LIN {X 0,Y 150.683,Z 393.041,A -85,B 0,C 180,E1 7413.083,E2 7413.083} C_VEL
LIN {X 0,Y 146.558,Z 378.59,A -85,B 0,C 180,E1 7406.767,E2 7406.767} C_VEL
LIN {X 0,Y 142.773,Z 366.039,A -85,B 0,C 180,E1 7400.503,E2 7400.503} C_VEL
LIN {X 0,Y 139.358,Z 355.664,A -85,B 0,C 180,E1 7394.549,E2 7394.549} C_VEL
LIN {X 0,Y 136.525,Z 347.614,A -85,B 0,C 180,E1 7389.278,E2 7389.278} C_VEL
LIN {X 0,Y 133.958,Z 340.934,A -85,B 0,C 180,E1 7384.287,E2 7384.287} C_VEL
LIN {X 0,Y 132.496,Z 337.338,A -85,B 0,C 180,E1 7381.303,E2 7381.303} C_VEL
LIN {X 0,Y 131.528,Z 334.4,A -85,B 0,C 180,E1 7378.699,E2 7378.699} C_VEL
LIN {X 0,Y 131.538,Z 334.397,A -85,B 0,C 180,E1 7371.703,E2 7371.703} C_VEL
LIN {X 0,Y 131.537,Z 334.414,A -85,B 0,C 180,E1 7364.864,E2 7364.864} C_VEL
LIN {X 0,Y 131.54,Z 334.399,A -85,B 0,C 180,E1 7358.015,E2 7358.015} C_VEL
LIN {X 0,Y 131.539,Z 334.371,A -85,B 0,C 180,E1 7350.936,E2 7350.936} C_VEL
LIN {X 0,Y 131.536,Z 334.411,A -85,B 0,C 180,E1 7344.184,E2 7344.184} C_VEL
LIN {X 0,Y 131.542,Z 334.371,A -85,B 0,C 180,E1 7337.439,E2 7337.439} C_VEL
LIN {X 0,Y 131.54,Z 334.396,A -85,B 0,C 180,E1 7330.537,E2 7330.537} C_VEL
LIN {X 0,Y 131.548,Z 334.386,A -85,B 0,C 180,E1 7323.696,E2 7323.696} C_VEL
LIN {X 0,Y 131.551,Z 334.382,A -85,B 0,C 180,E1 7317.128,E2 7317.128} C_VEL
LIN {X 0,Y 131.548,Z 334.403,A -85,B 0,C 180,E1 7310.461,E2 7310.461} C_VEL
LIN {X 0,Y 131.548,Z 334.375,A -85,B 0,C 180,E1 7303.625,E2 7303.625} C_VEL
LIN {X 0,Y 131.549,Z 334.398,A -85,B 0,C 180,E1 7296.543,E2 7296.543} C_VEL
LIN {X 0,Y 131.56,Z 334.411,A -85,B 0,C 180,E1 7289.561,E2 7289.561} C_VEL
LIN {X 0,Y 131.556,Z 334.412,A -85,B 0,C 180,E1 7282.573,E2 7282.573} C_VEL
LIN {X 0,Y 131.581,Z 334.588,A -85,B 0,C 180,E1 7280.814,E2 7280.814} C_VEL
LIN {X 0,Y 134.219,Z 341.466,A -85,B 0,C 180,E1 7274.883,E2 7274.883} C_VEL
LIN {X 0,Y 137.329,Z 350.554,A -85,B 0,C 180,E1 7268.2,E2 7268.2} C_VEL
LIN {X 0,Y 140.273,Z 360.105,A -85,B 0,C 180,E1 7262.098,E2 7262.098} C_VEL
LIN {X 0,Y 143.171,Z 370.927,A -85,B 0,C 180,E1 7256.031,E2 7256.031} C_VEL
LIN {X 0,Y 145.879,Z 382.116,A -85,B 0,C 180,E1 7250.396,E2 7250.396} C_VEL
LIN {X 0,Y 148.723,Z 395.438,A -85,B 0,C 180,E1 7244.353,E2 7244.353} C_VEL
LIN {X 0,Y 149.059,Z 398.299,A -85,B 0,C 180,E1 7243.164,E2 7243.164} C_VEL
LIN {X 0,Y 148.596,Z 421.413,A -85,B 0,C 180,E1 7240.916,E2 7240.916} C_VEL
LIN {X 0,Y 149.464,Z 452.011,A -85,B 0,C 180,E1 7237.85,E2 7237.85} C_VEL
LIN {X 0,Y 140.041,Z 546.315,A -85,B 0,C 180,E1 7229.401,E2 7229.401} C_VEL
LIN {X 0,Y 138.1,Z 565.524,A -85,B 0,C 180,E1 7226.897,E2 7226.897} C_VEL
LIN {X 0,Y 135.925,Z 584.105,A -85,B 0,C 180,E1 7223.627,E2 7223.627} C_VEL
LIN {X 0,Y 133.756,Z 602.389,A -85,B 0,C 180,E1 7219.423,E2 7219.423} C_VEL
LIN {X 0,Y 132.018,Z 618.485,A -85,B 0,C 180,E1 7214.691,E2 7214.691} C_VEL
LIN {X 0,Y 130.929,Z 632.317,A -85,B 0,C 180,E1 7209.665,E2 7209.665} C_VEL
LIN {X 0,Y 130.554,Z 645.192,A -85,B 0,C 180,E1 7203.946,E2 7203.946} C_VEL
LIN {X 0,Y 131.161,Z 656.496,A -85,B 0,C 180,E1 7197.809,E2 7197.809} C_VEL
LIN {X 0,Y 133.293,Z 666.98,A -85,B 0,C 180,E1 7190.931,E2 7190.931} C_VEL
LIN {X 0,Y 137.22,Z 675.28,A -85,B 0,C 180,E1 7184.354,E2 7184.354} C_VEL
LIN {X 0,Y 143.835,Z 682.507,A -85,B 0,C 180,E1 7177.516,E2 7177.516} C_VEL
LIN {X 0,Y 152.229,Z 687.511,A -85,B 0,C 180,E1 7171.663,E2 7171.663} C_VEL
LIN {X 0,Y 163.33,Z 691.005,A -85,B 0,C 180,E1 7166.141,E2 7166.141} C_VEL
LIN {X 0,Y 171.804,Z 692.342,A -85,B 0,C 180,E1 7162.878,E2 7162.878} C_VEL
LIN {X 0,Y 156.464,Z 696.456,A -85,B 0,C 180,E1 7156.764,E2 7156.764} C_VEL
LIN {X 0,Y 143.752,Z 699.352,A -85,B 0,C 180,E1 7148.759,E2 7148.759} C_VEL
LIN {X 0,Y 135.27,Z 700.716,A -85,B 0,C 180,E1 7139.202,E2 7139.202} C_VEL
LIN {X 0,Y 131.796,Z 700.428,A -85,B 0,C 180,E1 7129.043,E2 7129.043} C_VEL
LIN {X 0,Y 132.809,Z 698.4,A -85,B 0,C 180,E1 7119.1,E2 7119.1} C_VEL
LIN {X 0,Y 135.648,Z 695.5,A -85,B 0,C 180,E1 7112.115,E2 7112.115} C_VEL
LIN {X 0,Y 136.139,Z 694.711,A -85,B 0,C 180,E1 7110.845,E2 7110.845} C_VEL
LIN {X 0,Y 134.953,Z 689.744,A -85,B 0,C 180,E1 7106.18,E2 7106.18} C_VEL
LIN {X 0,Y 133.784,Z 681.429,A -85,B 0,C 180,E1 7100.105,E2 7100.105} C_VEL
LIN {X 0,Y 133.629,Z 670.856,A -85,B 0,C 180,E1 7093.931,E2 7093.931} C_VEL
LIN {X 0,Y 134.598,Z 658.65,A -85,B 0,C 180,E1 7088.2,E2 7088.2} C_VEL
LIN {X 0,Y 136.522,Z 644.855,A -85,B 0,C 180,E1 7082.998,E2 7082.998} C_VEL
LIN {X 0,Y 139.164,Z 629.313,A -85,B 0,C 180,E1 7078.37,E2 7078.37} C_VEL
LIN {X 0,Y 139.41,Z 627.91,A -85,B 0,C 180,E1 7078,E2 7078} C_VEL
LIN {X 0,Y 139.598,Z 621.253,A -85,B 0,C 180,E1 7076.361,E2 7076.361} C_VEL
LIN {X 0,Y 137.356,Z 608.461,A -85,B 0,C 180,E1 7073.628,E2 7073.628} C_VEL
LIN {X 0,Y 136.531,Z 599.282,A -85,B 0,C 180,E1 7071.919,E2 7071.919} C_VEL
LIN {X 0,Y 136.821,Z 596.182,A -85,B 0,C 180,E1 7071.399,E2 7071.399} C_VEL
LIN {X 0,Y 139.519,Z 577.848,A -85,B 0,C 180,E1 7068.757,E2 7068.757} C_VEL
LIN {X 0,Y 141.439,Z 558.683,A -85,B 0,C 180,E1 7066.782,E2 7066.782} C_VEL
LIN {X 0,Y 154.3,Z 431.413,A -85,B 0,C 180,E1 7057.035,E2 7057.035} C_VEL
LIN {X 0,Y 153.996,Z 422.024,A -85,B 0,C 180,E1 7056.193,E2 7056.193} C_VEL
LIN {X 0,Y 142.475,Z 393.084,A -85,B 0,C 180,E1 7051.528,E2 7051.528} C_VEL
LIN {X 0,Y 138.645,Z 379.476,A -85,B 0,C 180,E1 7045.187,E2 7045.187} C_VEL
LIN {X 0,Y 135.18,Z 367.855,A -85,B 0,C 180,E1 7038.999,E2 7038.999} C_VEL
LIN {X 0,Y 131.863,Z 357.589,A -85,B 0,C 180,E1 7032.709,E2 7032.709} C_VEL
LIN {X 0,Y 128.901,Z 349.101,A -85,B 0,C 180,E1 7026.688,E2 7026.688} C_VEL
LIN {X 0,Y 126.18,Z 342.172,A -85,B 0,C 180,E1 7020.915,E2 7020.915} C_VEL
LIN {X 0,Y 124.796,Z 338.717,A -85,B 0,C 180,E1 7017.711,E2 7017.711} C_VEL
LIN {X 0,Y 123.591,Z 335.399,A -85,B 0,C 180,E1 7014.274,E2 7014.274} C_VEL
LIN {X 0,Y 123.596,Z 335.388,A -85,B 0,C 180,E1 7007.391,E2 7007.391} C_VEL
LIN {X 0,Y 123.593,Z 335.369,A -85,B 0,C 180,E1 7000.636,E2 7000.636} C_VEL
LIN {X 0,Y 123.599,Z 335.38,A -85,B 0,C 180,E1 6993.59,E2 6993.59} C_VEL
LIN {X 0,Y 123.6,Z 335.394,A -85,B 0,C 180,E1 6986.423,E2 6986.423} C_VEL
LIN {X 0,Y 123.605,Z 335.352,A -85,B 0,C 180,E1 6979.073,E2 6979.073} C_VEL
LIN {X 0,Y 123.607,Z 335.396,A -85,B 0,C 180,E1 6971.922,E2 6971.922} C_VEL
LIN {X 0,Y 123.602,Z 335.357,A -85,B 0,C 180,E1 6965.049,E2 6965.049} C_VEL
LIN {X 0,Y 123.611,Z 335.38,A -85,B 0,C 180,E1 6957.975,E2 6957.975} C_VEL
LIN {X 0,Y 123.613,Z 335.386,A -85,B 0,C 180,E1 6950.845,E2 6950.845} C_VEL
LIN {X 0,Y 123.609,Z 335.362,A -85,B 0,C 180,E1 6943.563,E2 6943.563} C_VEL
LIN {X 0,Y 123.61,Z 335.385,A -85,B 0,C 180,E1 6936.499,E2 6936.499} C_VEL
LIN {X 0,Y 123.621,Z 335.399,A -85,B 0,C 180,E1 6929.533,E2 6929.533} C_VEL
LIN {X 0,Y 123.631,Z 335.526,A -85,B 0,C 180,E1 6925.125,E2 6925.125} C_VEL
LIN {X 0,Y 125.375,Z 340.333,A -85,B 0,C 180,E1 6920.356,E2 6920.356} C_VEL
LIN {X 0,Y 127.54,Z 345.72,A -85,B 0,C 180,E1 6915.468,E2 6915.468} C_VEL
LIN {X 0,Y 130.399,Z 354.265,A -85,B 0,C 180,E1 6908.873,E2 6908.873} C_VEL
LIN {X 0,Y 133.143,Z 363.456,A -85,B 0,C 180,E1 6902.733,E2 6902.733} C_VEL
LIN {X 0,Y 135.726,Z 373.257,A -85,B 0,C 180,E1 6896.962,E2 6896.962} C_VEL
LIN {X 0,Y 138.464,Z 384.941,A -85,B 0,C 180,E1 6890.81,E2 6890.81} C_VEL
LIN {X 0,Y 141.221,Z 398.27,A -85,B 0,C 180,E1 6884.492,E2 6884.492} C_VEL
LIN {X 0,Y 141.489,Z 400.719,A -85,B 0,C 180,E1 6884.143,E2 6884.143} C_VEL
LIN {X 0,Y 141.215,Z 429.3,A -85,B 0,C 180,E1 6881.261,E2 6881.261} C_VEL
LIN {X 0,Y 141.827,Z 452.369,A -85,B 0,C 180,E1 6878.82,E2 6878.82} C_VEL
LIN {X 0,Y 132.003,Z 547.522,A -85,B 0,C 180,E1 6869.752,E2 6869.752} C_VEL
LIN {X 0,Y 129.946,Z 567.105,A -85,B 0,C 180,E1 6866.991,E2 6866.991} C_VEL
LIN {X 0,Y 127.744,Z 585.451,A -85,B 0,C 180,E1 6863.519,E2 6863.519} C_VEL
LIN {X 0,Y 125.578,Z 603.516,A -85,B 0,C 180,E1 6859.046,E2 6859.046} C_VEL
LIN {X 0,Y 123.888,Z 619.491,A -85,B 0,C 180,E1 6854.005,E2 6854.005} C_VEL
LIN {X 0,Y 122.876,Z 633.784,A -85,B 0,C 180,E1 6848.415,E2 6848.415} C_VEL
LIN {X 0,Y 122.71,Z 646.517,A -85,B 0,C 180,E1 6842.328,E2 6842.328} C_VEL
LIN {X 0,Y 123.637,Z 657.727,A -85,B 0,C 180,E1 6835.82,E2 6835.82} C_VEL
LIN {X 0,Y 126.288,Z 668.167,A -85,B 0,C 180,E1 6828.578,E2 6828.578} C_VEL
LIN {X 0,Y 130.876,Z 676.512,A -85,B 0,C 180,E1 6821.74,E2 6821.74} C_VEL
LIN {X 0,Y 138.324,Z 683.804,A -85,B 0,C 180,E1 6814.75,E2 6814.75} C_VEL
LIN {X 0,Y 147.975,Z 689.161,A -85,B 0,C 180,E1 6808.643,E2 6808.643} C_VEL
LIN {X 0,Y 159.485,Z 692.66,A -85,B 0,C 180,E1 6803.44,E2 6803.44} C_VEL
LIN {X 0,Y 160.626,Z 692.942,A -85,B 0,C 180,E1 6802.92,E2 6802.92} C_VEL
LIN {X 0,Y 145.016,Z 696.125,A -85,B 0,C 180,E1 6795.816,E2 6795.816} C_VEL
LIN {X 0,Y 133.216,Z 697.907,A -85,B 0,C 180,E1 6786.905,E2 6786.905} C_VEL
LIN {X 0,Y 126.082,Z 698.177,A -85,B 0,C 180,E1 6776.336,E2 6776.336} C_VEL
LIN {X 0,Y 124.347,Z 696.755,A -85,B 0,C 180,E1 6765.205,E2 6765.205} C_VEL
LIN {X 0,Y 126.828,Z 693.769,A -85,B 0,C 180,E1 6755.432,E2 6755.432} C_VEL
LIN {X 0,Y 128.714,Z 691.564,A -85,B 0,C 180,E1 6751.116,E2 6751.116} C_VEL
LIN {X 0,Y 127.318,Z 685.883,A -85,B 0,C 180,E1 6745.908,E2 6745.908} C_VEL
LIN {X 0,Y 126.154,Z 677.072,A -85,B 0,C 180,E1 6739.5,E2 6739.5} C_VEL
LIN {X 0,Y 126.101,Z 666.701,A -85,B 0,C 180,E1 6733.418,E2 6733.418} C_VEL
LIN {X 0,Y 127.218,Z 653.846,A -85,B 0,C 180,E1 6727.353,E2 6727.353} C_VEL
LIN {X 0,Y 129.369,Z 639.086,A -85,B 0,C 180,E1 6721.783,E2 6721.783} C_VEL
LIN {X 0,Y 132.076,Z 623.504,A -85,B 0,C 180,E1 6717.182,E2 6717.182} C_VEL
LIN {X 0,Y 135.166,Z 605.997,A -85,B 0,C 180,E1 6713.193,E2 6713.193} C_VEL
LIN {X 0,Y 136.821,Z 596.182,A -85,B 0,C 180,E1 6711.399,E2 6711.399} C_VEL
LIN {X 0,Y 136.985,Z 589.005,A -85,B 0,C 180,E1 6710.233,E2 6710.233} C_VEL
LIN {X 0,Y 134.893,Z 577.488,A -85,B 0,C 180,E1 6708.509,E2 6708.509} C_VEL
LIN {X 0,Y 133.281,Z 567.956,A -85,B 0,C 180,E1 6707.256,E2 6707.256} C_VEL
LIN {X 0,Y 133.163,Z 562.543,A -85,B 0,C 180,E1 6706.673,E2 6706.673} C_VEL
LIN {X 0,Y 146.817,Z 431.575,A -85,B 0,C 180,E1 6695.935,E2 6695.935} C_VEL
LIN {X 0,Y 146.55,Z 424.082,A -85,B 0,C 180,E1 6695.212,E2 6695.212} C_VEL
LIN {X 0,Y 134.329,Z 393.285,A -85,B 0,C 180,E1 6689.921,E2 6689.921} C_VEL
LIN {X 0,Y 130.717,Z 380.305,A -85,B 0,C 180,E1 6683.444,E2 6683.444} C_VEL
LIN {X 0,Y 127.353,Z 368.889,A -85,B 0,C 180,E1 6676.894,E2 6676.894} C_VEL
LIN {X 0,Y 124.371,Z 359.459,A -85,B 0,C 180,E1 6670.662,E2 6670.662} C_VEL
LIN {X 0,Y 121.389,Z 350.875,A -85,B 0,C 180,E1 6664.021,E2 6664.021} C_VEL
LIN {X 0,Y 118.712,Z 343.91,A -85,B 0,C 180,E1 6657.593,E2 6657.593} C_VEL
LIN {X 0,Y 116.85,Z 339.701,A -85,B 0,C 180,E1 6652.984,E2 6652.984} C_VEL
LIN {X 0,Y 115.651,Z 336.365,A -85,B 0,C 180,E1 6649.043,E2 6649.043} C_VEL
LIN {X 0,Y 115.654,Z 336.359,A -85,B 0,C 180,E1 6641.875,E2 6641.875} C_VEL
LIN {X 0,Y 115.661,Z 336.386,A -85,B 0,C 180,E1 6634.947,E2 6634.947} C_VEL
LIN {X 0,Y 115.662,Z 336.365,A -85,B 0,C 180,E1 6627.599,E2 6627.599} C_VEL
LIN {X 0,Y 115.658,Z 336.343,A -85,B 0,C 180,E1 6620.239,E2 6620.239} C_VEL
LIN {X 0,Y 115.664,Z 336.388,A -85,B 0,C 180,E1 6612.723,E2 6612.723} C_VEL
LIN {X 0,Y 115.662,Z 336.342,A -85,B 0,C 180,E1 6605.389,E2 6605.389} C_VEL
LIN {X 0,Y 115.672,Z 336.369,A -85,B 0,C 180,E1 6598.172,E2 6598.172} C_VEL
LIN {X 0,Y 115.673,Z 336.373,A -85,B 0,C 180,E1 6590.752,E2 6590.752} C_VEL
LIN {X 0,Y 115.67,Z 336.35,A -85,B 0,C 180,E1 6583.493,E2 6583.493} C_VEL
LIN {X 0,Y 115.669,Z 336.37,A -85,B 0,C 180,E1 6576.317,E2 6576.317} C_VEL
LIN {X 0,Y 115.702,Z 336.586,A -85,B 0,C 180,E1 6570.244,E2 6570.244} C_VEL
LIN {X 0,Y 117.405,Z 340.903,A -85,B 0,C 180,E1 6565.111,E2 6565.111} C_VEL
LIN {X 0,Y 119.12,Z 345.515,A -85,B 0,C 180,E1 6560.332,E2 6560.332} C_VEL
LIN {X 0,Y 121.181,Z 351.079,A -85,B 0,C 180,E1 6555.177,E2 6555.177} C_VEL
LIN {X 0,Y 123.654,Z 358.59,A -85,B 0,C 180,E1 6549.155,E2 6549.155} C_VEL
LIN {X 0,Y 126.337,Z 367.948,A -85,B 0,C 180,E1 6542.672,E2 6542.672} C_VEL
LIN {X 0,Y 129.061,Z 378.829,A -85,B 0,C 180,E1 6536.093,E2 6536.093} C_VEL
LIN {X 0,Y 131.628,Z 390.58,A -85,B 0,C 180,E1 6529.78,E2 6529.78} C_VEL
LIN {X 0,Y 133.326,Z 398.795,A -85,B 0,C 180,E1 6525.886,E2 6525.886} C_VEL
LIN {X 0,Y 134.111,Z 402.002,A -85,B 0,C 180,E1 6525.384,E2 6525.384} C_VEL
LIN {X 0,Y 133.76,Z 432.444,A -85,B 0,C 180,E1 6522.122,E2 6522.122} C_VEL
LIN {X 0,Y 134.214,Z 452.567,A -85,B 0,C 180,E1 6519.865,E2 6519.865} C_VEL
LIN {X 0,Y 123.962,Z 548.599,A -85,B 0,C 180,E1 6510.114,E2 6510.114} C_VEL
LIN {X 0,Y 121.85,Z 568.006,A -85,B 0,C 180,E1 6507.166,E2 6507.166} C_VEL
LIN {X 0,Y 119.58,Z 586.534,A -85,B 0,C 180,E1 6503.393,E2 6503.393} C_VEL
LIN {X 0,Y 117.421,Z 604.445,A -85,B 0,C 180,E1 6498.614,E2 6498.614} C_VEL
LIN {X 0,Y 115.734,Z 620.989,A -85,B 0,C 180,E1 6492.973,E2 6492.973} C_VEL
LIN {X 0,Y 114.891,Z 635.095,A -85,B 0,C 180,E1 6486.991,E2 6486.991} C_VEL
LIN {X 0,Y 114.992,Z 648.101,A -85,B 0,C 180,E1 6480.267,E2 6480.267} C_VEL
LIN {X 0,Y 116.418,Z 659.541,A -85,B 0,C 180,E1 6473.087,E2 6473.087} C_VEL
LIN {X 0,Y 119.971,Z 670.222,A -85,B 0,C 180,E1 6465.199,E2 6465.199} C_VEL
LIN {X 0,Y 126.061,Z 679.001,A -85,B 0,C 180,E1 6457.616,E2 6457.616} C_VEL
LIN {X 0,Y 134.788,Z 686.098,A -85,B 0,C 180,E1 6450.68,E2 6450.68} C_VEL
LIN {X 0,Y 145.748,Z 691.316,A -85,B 0,C 180,E1 6444.727,E2 6444.727} C_VEL
LIN {X 0,Y 149.723,Z 692.688,A -85,B 0,C 180,E1 6442.947,E2 6442.947} C_VEL
LIN {X 0,Y 134.373,Z 694.869,A -85,B 0,C 180,E1 6434.987,E2 6434.987} C_VEL
LIN {X 0,Y 123.091,Z 695.657,A -85,B 0,C 180,E1 6424.657,E2 6424.657} C_VEL
LIN {X 0,Y 117.454,Z 694.796,A -85,B 0,C 180,E1 6412.528,E2 6412.528} C_VEL
LIN {X 0,Y 117.805,Z 692.214,A -85,B 0,C 180,E1 6400.765,E2 6400.765} C_VEL
LIN {X 0,Y 121.084,Z 688.699,A -85,B 0,C 180,E1 6392.2,E2 6392.2} C_VEL
LIN {X 0,Y 121.333,Z 688.211,A -85,B 0,C 180,E1 6391.42,E2 6391.42} C_VEL
LIN {X 0,Y 119.736,Z 681.874,A -85,B 0,C 180,E1 6385.694,E2 6385.694} C_VEL
LIN {X 0,Y 118.584,Z 672.386,A -85,B 0,C 180,E1 6378.822,E2 6378.822} C_VEL
LIN {X 0,Y 118.696,Z 660.99,A -85,B 0,C 180,E1 6372.171,E2 6372.171} C_VEL
LIN {X 0,Y 120.042,Z 647.588,A -85,B 0,C 180,E1 6365.916,E2 6365.916} C_VEL
LIN {X 0,Y 122.349,Z 632.67,A -85,B 0,C 180,E1 6360.373,E2 6360.373} C_VEL
LIN {X 0,Y 125.179,Z 616.642,A -85,B 0,C 180,E1 6355.733,E2 6355.733} C_VEL
LIN {X 0,Y 128.43,Z 598.059,A -85,B 0,C 180,E1 6351.65,E2 6351.65} C_VEL
LIN {X 0,Y 131.193,Z 580.337,A -85,B 0,C 180,E1 6348.77,E2 6348.77} C_VEL
LIN {X 0,Y 133.163,Z 562.543,A -85,B 0,C 180,E1 6346.673,E2 6346.673} C_VEL
LIN {X 0,Y 133.015,Z 556.072,A -85,B 0,C 180,E1 6346.003,E2 6346.003} C_VEL
LIN {X 0,Y 128.539,Z 534.863,A -85,B 0,C 180,E1 6343.589,E2 6343.589} C_VEL
LIN {X 0,Y 128.454,Z 528.37,A -85,B 0,C 180,E1 6342.932,E2 6342.932} C_VEL
LIN {X 0,Y 139.344,Z 431.761,A -85,B 0,C 180,E1 6334.772,E2 6334.772} C_VEL
LIN {X 0,Y 139.105,Z 426.223,A -85,B 0,C 180,E1 6334.195,E2 6334.195} C_VEL
LIN {X 0,Y 126.823,Z 395.218,A -85,B 0,C 180,E1 6328.623,E2 6328.623} C_VEL
LIN {X 0,Y 126.173,Z 393.363,A -85,B 0,C 180,E1 6328.139,E2 6328.139} C_VEL
LIN {X 0,Y 122.795,Z 381.062,A -85,B 0,C 180,E1 6321.501,E2 6321.501} C_VEL
LIN {X 0,Y 119.76,Z 370.576,A -85,B 0,C 180,E1 6315.006,E2 6315.006} C_VEL
LIN {X 0,Y 116.863,Z 361.306,A -85,B 0,C 180,E1 6308.37,E2 6308.37} C_VEL
LIN {X 0,Y 114.203,Z 353.818,A -85,B 0,C 180,E1 6302.014,E2 6302.014} C_VEL
LIN {X 0,Y 112.073,Z 348.172,A -85,B 0,C 180,E1 6296.427,E2 6296.427} C_VEL
LIN {X 0,Y 110.565,Z 344.518,A -85,B 0,C 180,E1 6292.212,E2 6292.212} C_VEL
LIN {X 0,Y 109.183,Z 341.077,A -85,B 0,C 180,E1 6287.849,E2 6287.849} C_VEL
LIN {X 0,Y 107.714,Z 337.348,A -85,B 0,C 180,E1 6282.171,E2 6282.171} C_VEL
LIN {X 0,Y 107.719,Z 337.369,A -85,B 0,C 180,E1 6274.733,E2 6274.733} C_VEL
LIN {X 0,Y 107.721,Z 337.354,A -85,B 0,C 180,E1 6267.438,E2 6267.438} C_VEL
LIN {X 0,Y 107.72,Z 337.33,A -85,B 0,C 180,E1 6260.185,E2 6260.185} C_VEL
LIN {X 0,Y 107.725,Z 337.377,A -85,B 0,C 180,E1 6252.647,E2 6252.647} C_VEL
LIN {X 0,Y 107.721,Z 337.331,A -85,B 0,C 180,E1 6245.128,E2 6245.128} C_VEL
LIN {X 0,Y 107.732,Z 337.347,A -85,B 0,C 180,E1 6237.644,E2 6237.644} C_VEL
LIN {X 0,Y 107.731,Z 337.37,A -85,B 0,C 180,E1 6230.08,E2 6230.08} C_VEL
LIN {X 0,Y 107.726,Z 337.341,A -85,B 0,C 180,E1 6222.322,E2 6222.322} C_VEL
LIN {X 0,Y 107.757,Z 337.496,A -85,B 0,C 180,E1 6216.924,E2 6216.924} C_VEL
LIN {X 0,Y 109.659,Z 342.262,A -85,B 0,C 180,E1 6209.996,E2 6209.996} C_VEL
LIN {X 0,Y 111.275,Z 346.435,A -85,B 0,C 180,E1 6204.841,E2 6204.841} C_VEL
LIN {X 0,Y 113.279,Z 351.544,A -85,B 0,C 180,E1 6199.314,E2 6199.314} C_VEL
LIN {X 0,Y 115.579,Z 358.645,A -85,B 0,C 180,E1 6192.891,E2 6192.891} C_VEL
LIN {X 0,Y 118.006,Z 366.771,A -85,B 0,C 180,E1 6186.529,E2 6186.529} C_VEL
LIN {X 0,Y 120.432,Z 376.228,A -85,B 0,C 180,E1 6180.119,E2 6180.119} C_VEL
LIN {X 0,Y 122.91,Z 387.17,A -85,B 0,C 180,E1 6173.565,E2 6173.565} C_VEL
LIN {X 0,Y 125.238,Z 398.592,A -85,B 0,C 180,E1 6167.571,E2 6167.571} C_VEL
LIN {X 0,Y 126.703,Z 403.867,A -85,B 0,C 180,E1 6166.638,E2 6166.638} C_VEL
LIN {X 0,Y 126.314,Z 436.525,A -85,B 0,C 180,E1 6162.912,E2 6162.912} C_VEL
LIN {X 0,Y 126.593,Z 452.849,A -85,B 0,C 180,E1 6160.972,E2 6160.972} C_VEL
LIN {X 0,Y 115.932,Z 549.42,A -85,B 0,C 180,E1 6150.502,E2 6150.502} C_VEL
LIN {X 0,Y 113.767,Z 568.67,A -85,B 0,C 180,E1 6147.355,E2 6147.355} C_VEL
LIN {X 0,Y 111.434,Z 587.368,A -85,B 0,C 180,E1 6143.245,E2 6143.245} C_VEL
LIN {X 0,Y 109.285,Z 605.173,A -85,B 0,C 180,E1 6138.115,E2 6138.115} C_VEL
LIN {X 0,Y 107.679,Z 621.647,A -85,B 0,C 180,E1 6132.051,E2 6132.051} C_VEL
LIN {X 0,Y 106.992,Z 635.726,A -85,B 0,C 180,E1 6125.623,E2 6125.623} C_VEL
LIN {X 0,Y 107.362,Z 648.727,A -85,B 0,C 180,E1 6118.391,E2 6118.391} C_VEL
LIN {X 0,Y 109.103,Z 659.821,A -85,B 0,C 180,E1 6111.03,E2 6111.03} C_VEL
LIN {X 0,Y 113.366,Z 670.807,A -85,B 0,C 180,E1 6102.543,E2 6102.543} C_VEL
LIN {X 0,Y 120.072,Z 679.619,A -85,B 0,C 180,E1 6094.862,E2 6094.862} C_VEL
LIN {X 0,Y 129.605,Z 686.899,A -85,B 0,C 180,E1 6087.832,E2 6087.832} C_VEL
LIN {X 0,Y 138.917,Z 691.55,A -85,B 0,C 180,E1 6082.862,E2 6082.862} C_VEL
LIN {X 0,Y 123.982,Z 692.77,A -85,B 0,C 180,E1 6073.916,E2 6073.916} C_VEL
LIN {X 0,Y 113.782,Z 692.575,A -85,B 0,C 180,E1 6062.419,E2 6062.419} C_VEL
LIN {X 0,Y 109.855,Z 690.815,A -85,B 0,C 180,E1 6049.684,E2 6049.684} C_VEL
LIN {X 0,Y 111.613,Z 687.451,A -85,B 0,C 180,E1 6037.726,E2 6037.726} C_VEL
LIN {X 0,Y 114.056,Z 684.889,A -85,B 0,C 180,E1 6032.013,E2 6032.013} C_VEL
LIN {X 0,Y 112.28,Z 678.232,A -85,B 0,C 180,E1 6025.919,E2 6025.919} C_VEL
LIN {X 0,Y 111.109,Z 668.549,A -85,B 0,C 180,E1 6018.81,E2 6018.81} C_VEL
LIN {X 0,Y 111.271,Z 656.529,A -85,B 0,C 180,E1 6011.673,E2 6011.673} C_VEL
LIN {X 0,Y 112.716,Z 642.741,A -85,B 0,C 180,E1 6005.084,E2 6005.084} C_VEL
LIN {X 0,Y 115.092,Z 627.717,A -85,B 0,C 180,E1 5999.459,E2 5999.459} C_VEL
LIN {X 0,Y 118.083,Z 610.852,A -85,B 0,C 180,E1 5994.553,E2 5994.553} C_VEL
LIN {X 0,Y 121.13,Z 593.331,A -85,B 0,C 180,E1 5990.71,E2 5990.71} C_VEL
LIN {X 0,Y 123.885,Z 574.95,A -85,B 0,C 180,E1 5987.725,E2 5987.725} C_VEL
LIN {X 0,Y 125.894,Z 555.13,A -85,B 0,C 180,E1 5985.467,E2 5985.467} C_VEL
LIN {X 0,Y 128.454,Z 528.37,A -85,B 0,C 180,E1 5982.932,E2 5982.932} C_VEL
LIN {X 0,Y 128.286,Z 520.81,A -85,B 0,C 180,E1 5982.145,E2 5982.145} C_VEL
LIN {X 0,Y 124.387,Z 500.678,A -85,B 0,C 180,E1 5979.616,E2 5979.616} C_VEL
LIN {X 0,Y 124.362,Z 494.19,A -85,B 0,C 180,E1 5978.92,E2 5978.92} C_VEL
LIN {X 0,Y 131.888,Z 431.825,A -85,B 0,C 180,E1 5973.518,E2 5973.518} C_VEL
LIN {X 0,Y 131.622,Z 428.233,A -85,B 0,C 180,E1 5973.099,E2 5973.099} C_VEL
LIN {X 0,Y 119.491,Z 397.209,A -85,B 0,C 180,E1 5967.139,E2 5967.139} C_VEL
LIN {X 0,Y 118.165,Z 393.866,A -85,B 0,C 180,E1 5966.381,E2 5966.381} C_VEL
LIN {X 0,Y 114.905,Z 381.743,A -85,B 0,C 180,E1 5959.316,E2 5959.316} C_VEL
LIN {X 0,Y 111.969,Z 371.508,A -85,B 0,C 180,E1 5952.382,E2 5952.382} C_VEL
LIN {X 0,Y 109.197,Z 362.498,A -85,B 0,C 180,E1 5945.261,E2 5945.261} C_VEL
LIN {X 0,Y 106.608,Z 355.349,A -85,B 0,C 180,E1 5938.395,E2 5938.395} C_VEL
LIN {X 0,Y 104.82,Z 350.243,A -85,B 0,C 180,E1 5932.727,E2 5932.727} C_VEL
LIN {X 0,Y 103.061,Z 346.148,A -85,B 0,C 180,E1 5927.115,E2 5927.115} C_VEL
LIN {X 0,Y 101.468,Z 342.343,A -85,B 0,C 180,E1 5921.033,E2 5921.033} C_VEL
LIN {X 0,Y 99.78,Z 338.329,A -85,B 0,C 180,E1 5912.562,E2 5912.562} C_VEL
LIN {X 0,Y 99.78,Z 338.368,A -85,B 0,C 180,E1 5905.179,E2 5905.179} C_VEL
LIN {X 0,Y 99.782,Z 338.317,A -85,B 0,C 180,E1 5897.839,E2 5897.839} C_VEL
LIN {X 0,Y 99.786,Z 338.33,A -85,B 0,C 180,E1 5889.882,E2 5889.882} C_VEL
LIN {X 0,Y 99.791,Z 338.353,A -85,B 0,C 180,E1 5882.07,E2 5882.07} C_VEL
LIN {X 0,Y 99.785,Z 338.317,A -85,B 0,C 180,E1 5874.252,E2 5874.252} C_VEL
LIN {X 0,Y 99.817,Z 338.544,A -85,B 0,C 180,E1 5866.284,E2 5866.284} C_VEL
LIN {X 0,Y 101.816,Z 343.21,A -85,B 0,C 180,E1 5856.763,E2 5856.763} C_VEL
LIN {X 0,Y 103.466,Z 347.241,A -85,B 0,C 180,E1 5850.549,E2 5850.549} C_VEL
LIN {X 0,Y 105.024,Z 351.471,A -85,B 0,C 180,E1 5845.081,E2 5845.081} C_VEL
LIN {X 0,Y 106.803,Z 356.21,A -85,B 0,C 180,E1 5839.75,E2 5839.75} C_VEL
LIN {X 0,Y 109.236,Z 364.002,A -85,B 0,C 180,E1 5832.415,E2 5832.415} C_VEL
LIN {X 0,Y 111.566,Z 372.505,A -85,B 0,C 180,E1 5825.649,E2 5825.649} C_VEL
LIN {X 0,Y 113.905,Z 382.437,A -85,B 0,C 180,E1 5818.804,E2 5818.804} C_VEL
LIN {X 0,Y 116.218,Z 393.551,A -85,B 0,C 180,E1 5812.034,E2 5812.034} C_VEL
LIN {X 0,Y 117.196,Z 398.468,A -85,B 0,C 180,E1 5809.414,E2 5809.414} C_VEL
LIN {X 0,Y 119.342,Z 405.588,A -85,B 0,C 180,E1 5808.024,E2 5808.024} C_VEL
LIN {X 0,Y 118.877,Z 440.87,A -85,B 0,C 180,E1 5803.712,E2 5803.712} C_VEL
LIN {X 0,Y 118.967,Z 453.25,A -85,B 0,C 180,E1 5802.158,E2 5802.158} C_VEL
LIN {X 0,Y 107.925,Z 549.879,A -85,B 0,C 180,E1 5790.933,E2 5790.933} C_VEL
LIN {X 0,Y 105.723,Z 568.92,A -85,B 0,C 180,E1 5787.598,E2 5787.598} C_VEL
LIN {X 0,Y 103.321,Z 587.877,A -85,B 0,C 180,E1 5783.095,E2 5783.095} C_VEL
LIN {X 0,Y 101.214,Z 605.379,A -85,B 0,C 180,E1 5777.644,E2 5777.644} C_VEL
LIN {X 0,Y 99.717,Z 621.49,A -85,B 0,C 180,E1 5771.267,E2 5771.267} C_VEL
LIN {X 0,Y 99.17,Z 636.206,A -85,B 0,C 180,E1 5764.039,E2 5764.039} C_VEL
LIN {X 0,Y 99.915,Z 649.606,A -85,B 0,C 180,E1 5755.975,E2 5755.975} C_VEL
LIN {X 0,Y 102.184,Z 660.678,A -85,B 0,C 180,E1 5748.134,E2 5748.134} C_VEL
LIN {X 0,Y 107.285,Z 671.655,A -85,B 0,C 180,E1 5739.251,E2 5739.251} C_VEL
LIN {X 0,Y 114.916,Z 680.567,A -85,B 0,C 180,E1 5731.402,E2 5731.402} C_VEL
LIN {X 0,Y 125.507,Z 688.043,A -85,B 0,C 180,E1 5724.355,E2 5724.355} C_VEL
LIN {X 0,Y 128.463,Z 689.668,A -85,B 0,C 180,E1 5722.74,E2 5722.74} C_VEL
LIN {X 0,Y 113.675,Z 689.994,A -85,B 0,C 180,E1 5712.358,E2 5712.358} C_VEL
LIN {X 0,Y 104.72,Z 688.78,A -85,B 0,C 180,E1 5699.145,E2 5699.145} C_VEL
LIN {X 0,Y 102.918,Z 685.964,A -85,B 0,C 180,E1 5685.211,E2 5685.211} C_VEL
LIN {X 0,Y 106.224,Z 681.865,A -85,B 0,C 180,E1 5673.747,E2 5673.747} C_VEL
LIN {X 0,Y 106.735,Z 681.177,A -85,B 0,C 180,E1 5672.42,E2 5672.42} C_VEL
LIN {X 0,Y 104.743,Z 673.676,A -85,B 0,C 180,E1 5665.624,E2 5665.624} C_VEL
LIN {X 0,Y 103.64,Z 663.803,A -85,B 0,C 180,E1 5658.316,E2 5658.316} C_VEL
LIN {X 0,Y 103.911,Z 651.48,A -85,B 0,C 180,E1 5650.908,E2 5650.908} C_VEL
LIN {X 0,Y 105.531,Z 637.096,A -85,B 0,C 180,E1 5643.978,E2 5643.978} C_VEL
LIN {X 0,Y 107.892,Z 622.458,A -85,B 0,C 180,E1 5638.431,E2 5638.431} C_VEL
LIN {X 0,Y 110.907,Z 605.533,A -85,B 0,C 180,E1 5633.492,E2 5633.492} C_VEL
LIN {X 0,Y 113.998,Z 587.598,A -85,B 0,C 180,E1 5629.536,E2 5629.536} C_VEL
LIN {X 0,Y 116.496,Z 569.711,A -85,B 0,C 180,E1 5626.685,E2 5626.685} C_VEL
LIN {X 0,Y 119.937,Z 534.705,A -85,B 0,C 180,E1 5622.859,E2 5622.859} C_VEL
LIN {X 0,Y 124.362,Z 494.19,A -85,B 0,C 180,E1 5618.92,E2 5618.92} C_VEL
LIN {X 0,Y 124.26,Z 486.631,A -85,B 0,C 180,E1 5618.095,E2 5618.095} C_VEL
LIN {X 0,Y 120.782,Z 466.491,A -85,B 0,C 180,E1 5615.383,E2 5615.383} C_VEL
LIN {X 0,Y 120.91,Z 460.005,A -85,B 0,C 180,E1 5614.677,E2 5614.677} C_VEL
LIN {X 0,Y 124.456,Z 431.855,A -85,B 0,C 180,E1 5612.165,E2 5612.165} C_VEL
LIN {X 0,Y 122.62,Z 426.226,A -85,B 0,C 180,E1 5611.181,E2 5611.181} C_VEL
LIN {X 0,Y 111.372,Z 397.297,A -85,B 0,C 180,E1 5605.085,E2 5605.085} C_VEL
LIN {X 0,Y 110.023,Z 393.836,A -85,B 0,C 180,E1 5604.146,E2 5604.146} C_VEL
LIN {X 0,Y 107.025,Z 382.378,A -85,B 0,C 180,E1 5596.842,E2 5596.842} C_VEL
LIN {X 0,Y 104.224,Z 372.408,A -85,B 0,C 180,E1 5589.394,E2 5589.394} C_VEL
LIN {X 0,Y 101.729,Z 364.319,A -85,B 0,C 180,E1 5582.261,E2 5582.261} C_VEL
LIN {X 0,Y 99.506,Z 357.893,A -85,B 0,C 180,E1 5575.398,E2 5575.398} C_VEL
LIN {X 0,Y 97.873,Z 353.728,A -85,B 0,C 180,E1 5570.007,E2 5570.007} C_VEL
LIN {X 0,Y 96.829,Z 351.02,A -85,B 0,C 180,E1 5566.062,E2 5566.062} C_VEL
LIN {X 0,Y 95.52,Z 347.649,A -85,B 0,C 180,E1 5560.389,E2 5560.389} C_VEL
LIN {X 0,Y 93.825,Z 343.661,A -85,B 0,C 180,E1 5551.355,E2 5551.355} C_VEL
LIN {X 0,Y 92.256,Z 341.032,A -85,B 0,C 180,E1 5540.263,E2 5540.263} C_VEL
LIN {X 0,Y 91.984,Z 340.132,A -85,B 0,C 180,E1 5532.356,E2 5532.356} C_VEL
LIN {X 0,Y 92.007,Z 340.214,A -85,B 0,C 180,E1 5525.161,E2 5525.161} C_VEL
LIN {X 0,Y 92.479,Z 341.58,A -85,B 0,C 180,E1 5516.207,E2 5516.207} C_VEL
LIN {X 0,Y 94.032,Z 344.064,A -85,B 0,C 180,E1 5506.679,E2 5506.679} C_VEL
LIN {X 0,Y 95.827,Z 348.515,A -85,B 0,C 180,E1 5497.188,E2 5497.188} C_VEL
LIN {X 0,Y 97.26,Z 352.184,A -85,B 0,C 180,E1 5491.174,E2 5491.174} C_VEL
LIN {X 0,Y 98.777,Z 356.501,A -85,B 0,C 180,E1 5485.351,E2 5485.351} C_VEL
LIN {X 0,Y 100.769,Z 362.445,A -85,B 0,C 180,E1 5478.55,E2 5478.55} C_VEL
LIN {X 0,Y 102.812,Z 369.439,A -85,B 0,C 180,E1 5471.864,E2 5471.864} C_VEL
LIN {X 0,Y 105.024,Z 378.197,A -85,B 0,C 180,E1 5464.725,E2 5464.725} C_VEL
LIN {X 0,Y 107.133,Z 387.904,A -85,B 0,C 180,E1 5457.857,E2 5457.857} C_VEL
LIN {X 0,Y 109.189,Z 398.337,A -85,B 0,C 180,E1 5451.483,E2 5451.483} C_VEL
LIN {X 0,Y 111.983,Z 407.566,A -85,B 0,C 180,E1 5449.486,E2 5449.486} C_VEL
LIN {X 0,Y 111.438,Z 445.078,A -85,B 0,C 180,E1 5444.576,E2 5444.576} C_VEL
LIN {X 0,Y 111.374,Z 453.531,A -85,B 0,C 180,E1 5443.46,E2 5443.46} C_VEL
LIN {X 0,Y 99.921,Z 550.213,A -85,B 0,C 180,E1 5431.387,E2 5431.387} C_VEL
LIN {X 0,Y 97.638,Z 569.39,A -85,B 0,C 180,E1 5427.761,E2 5427.761} C_VEL
LIN {X 0,Y 95.081,Z 589.319,A -85,B 0,C 180,E1 5422.561,E2 5422.561} C_VEL
LIN {X 0,Y 93.019,Z 606.833,A -85,B 0,C 180,E1 5416.54,E2 5416.54} C_VEL
LIN {X 0,Y 91.691,Z 623.094,A -85,B 0,C 180,E1 5409.405,E2 5409.405} C_VEL
LIN {X 0,Y 91.486,Z 637.554,A -85,B 0,C 180,E1 5401.557,E2 5401.557} C_VEL
LIN {X 0,Y 92.673,Z 650.334,A -85,B 0,C 180,E1 5393.175,E2 5393.175} C_VEL
LIN {X 0,Y 95.848,Z 662.095,A -85,B 0,C 180,E1 5384.254,E2 5384.254} C_VEL
LIN {X 0,Y 102.055,Z 672.967,A -85,B 0,C 180,E1 5375.076,E2 5375.076} C_VEL
LIN {X 0,Y 111.403,Z 682.341,A -85,B 0,C 180,E1 5366.798,E2 5366.798} C_VEL
LIN {X 0,Y 118.22,Z 687.037,A -85,B 0,C 180,E1 5362.479,E2 5362.479} C_VEL
LIN {X 0,Y 104.113,Z 686.46,A -85,B 0,C 180,E1 5350.777,E2 5350.777} C_VEL
LIN {X 0,Y 96.575,Z 684.282,A -85,B 0,C 180,E1 5335.779,E2 5335.779} C_VEL
LIN {X 0,Y 96.736,Z 680.655,A -85,B 0,C 180,E1 5321.33,E2 5321.33} C_VEL
LIN {X 0,Y 99.567,Z 677.444,A -85,B 0,C 180,E1 5313.17,E2 5313.17} C_VEL
LIN {X 0,Y 97.296,Z 669.074,A -85,B 0,C 180,E1 5305.516,E2 5305.516} C_VEL
LIN {X 0,Y 96.219,Z 658.189,A -85,B 0,C 180,E1 5297.4,E2 5297.4} C_VEL
LIN {X 0,Y 96.653,Z 645.549,A -85,B 0,C 180,E1 5289.728,E2 5289.728} C_VEL
LIN {X 0,Y 98.402,Z 631.203,A -85,B 0,C 180,E1 5282.796,E2 5282.796} C_VEL
LIN {X 0,Y 101.079,Z 615.078,A -85,B 0,C 180,E1 5276.707,E2 5276.707} C_VEL
LIN {X 0,Y 104.144,Z 597.844,A -85,B 0,C 180,E1 5271.8,E2 5271.8} C_VEL
LIN {X 0,Y 107.15,Z 579.815,A -85,B 0,C 180,E1 5267.975,E2 5267.975} C_VEL
LIN {X 0,Y 109.394,Z 561.32,A -85,B 0,C 180,E1 5265.204,E2 5265.204} C_VEL
LIN {X 0,Y 120.91,Z 460.005,A -85,B 0,C 180,E1 5254.677,E2 5254.677} C_VEL
LIN {X 0,Y 121.103,Z 451.315,A -85,B 0,C 180,E1 5253.723,E2 5253.723} C_VEL
LIN {X 0,Y 119.524,Z 441.782,A -85,B 0,C 180,E1 5252.344,E2 5252.344} C_VEL
LIN {X 0,Y 115.274,Z 428.543,A -85,B 0,C 180,E1 5249.936,E2 5249.936} C_VEL
LIN {X 0,Y 114.528,Z 426.555,A -85,B 0,C 180,E1 5249.533,E2 5249.533} C_VEL
LIN {X 0,Y 104.345,Z 400.037,A -85,B 0,C 180,E1 5243.478,E2 5243.478} C_VEL
LIN {X 0,Y 102.017,Z 394.143,A -85,B 0,C 180,E1 5241.874,E2 5241.874} C_VEL
LIN {X 0,Y 99.373,Z 383.736,A -85,B 0,C 180,E1 5234.577,E2 5234.577} C_VEL
LIN {X 0,Y 96.897,Z 374.616,A -85,B 0,C 180,E1 5227.121,E2 5227.121} C_VEL
LIN {X 0,Y 94.681,Z 367.287,A -85,B 0,C 180,E1 5220.009,E2 5220.009} C_VEL
LIN {X 0,Y 92.672,Z 361.324,A -85,B 0,C 180,E1 5212.988,E2 5212.988} C_VEL
LIN {X 0,Y 90.82,Z 356.254,A -85,B 0,C 180,E1 5205.632,E2 5205.632} C_VEL
LIN {X 0,Y 89.573,Z 352.935,A -85,B 0,C 180,E1 5199.646,E2 5199.646} C_VEL
LIN {X 0,Y 88.084,Z 349.218,A -85,B 0,C 180,E1 5190.796,E2 5190.796} C_VEL
LIN {X 0,Y 86.652,Z 346.587,A -85,B 0,C 180,E1 5178.888,E2 5178.888} C_VEL
LIN {X 0,Y 86.456,Z 345.832,A -85,B 0,C 180,E1 5170.262,E2 5170.262} C_VEL
LIN {X 0,Y 86.547,Z 346.308,A -85,B 0,C 180,E1 5162.524,E2 5162.524} C_VEL
LIN {X 0,Y 87.267,Z 348.07,A -85,B 0,C 180,E1 5152.921,E2 5152.921} C_VEL
LIN {X 0,Y 88.256,Z 349.585,A -85,B 0,C 180,E1 5147.126,E2 5147.126} C_VEL
LIN {X 0,Y 89.823,Z 353.791,A -85,B 0,C 180,E1 5137.671,E2 5137.671} C_VEL
LIN {X 0,Y 91.162,Z 357.554,A -85,B 0,C 180,E1 5131.252,E2 5131.252} C_VEL
LIN {X 0,Y 92.876,Z 362.388,A -85,B 0,C 180,E1 5124.435,E2 5124.435} C_VEL
LIN {X 0,Y 94.905,Z 369.319,A -85,B 0,C 180,E1 5116.594,E2 5116.594} C_VEL
LIN {X 0,Y 96.842,Z 376.906,A -85,B 0,C 180,E1 5109.444,E2 5109.444} C_VEL
LIN {X 0,Y 98.8,Z 385.808,A -85,B 0,C 180,E1 5102.251,E2 5102.251} C_VEL
LIN {X 0,Y 100.808,Z 396.247,A -85,B 0,C 180,E1 5094.876,E2 5094.876} C_VEL
LIN {X 0,Y 101.246,Z 398.326,A -85,B 0,C 180,E1 5093.746,E2 5093.746} C_VEL
LIN {X 0,Y 104.68,Z 409.264,A -85,B 0,C 180,E1 5091.132,E2 5091.132} C_VEL
LIN {X 0,Y 103.975,Z 447.961,A -85,B 0,C 180,E1 5085.697,E2 5085.697} C_VEL
LIN {X 0,Y 103.763,Z 454.07,A -85,B 0,C 180,E1 5084.86,E2 5084.86} C_VEL
LIN {X 0,Y 91.879,Z 550.769,A -85,B 0,C 180,E1 5071.806,E2 5071.806} C_VEL
LIN {X 0,Y 89.42,Z 570.758,A -85,B 0,C 180,E1 5067.637,E2 5067.637} C_VEL
LIN {X 0,Y 87.001,Z 589.468,A -85,B 0,C 180,E1 5062.277,E2 5062.277} C_VEL
LIN {X 0,Y 84.91,Z 607.749,A -85,B 0,C 180,E1 5055.353,E2 5055.353} C_VEL
LIN {X 0,Y 83.806,Z 623.866,A -85,B 0,C 180,E1 5047.531,E2 5047.531} C_VEL
LIN {X 0,Y 83.957,Z 638.221,A -85,B 0,C 180,E1 5038.967,E2 5038.967} C_VEL
LIN {X 0,Y 85.89,Z 651.759,A -85,B 0,C 180,E1 5029.256,E2 5029.256} C_VEL
LIN {X 0,Y 90.018,Z 663.363,A -85,B 0,C 180,E1 5019.85,E2 5019.85} C_VEL
LIN {X 0,Y 97.436,Z 674.159,A -85,B 0,C 180,E1 5010.482,E2 5010.482} C_VEL
LIN {X 0,Y 108.264,Z 683.747,A -85,B 0,C 180,E1 5002.075,E2 5002.075} C_VEL
LIN {X 0,Y 94.918,Z 682.337,A -85,B 0,C 180,E1 4988.772,E2 4988.772} C_VEL
LIN {X 0,Y 89.187,Z 679.336,A -85,B 0,C 180,E1 4972.411,E2 4972.411} C_VEL
LIN {X 0,Y 91.087,Z 674.992,A -85,B 0,C 180,E1 4957.574,E2 4957.574} C_VEL
LIN {X 0,Y 92.449,Z 673.547,A -85,B 0,C 180,E1 4954.036,E2 4954.036} C_VEL
LIN {X 0,Y 90.061,Z 665.136,A -85,B 0,C 180,E1 4946.185,E2 4946.185} C_VEL
LIN {X 0,Y 88.899,Z 654.086,A -85,B 0,C 180,E1 4937.666,E2 4937.666} C_VEL
LIN {X 0,Y 89.326,Z 640.922,A -85,B 0,C 180,E1 4929.359,E2 4929.359} C_VEL
LIN {X 0,Y 91.086,Z 626.648,A -85,B 0,C 180,E1 4922.197,E2 4922.197} C_VEL
LIN {X 0,Y 93.916,Z 609.717,A -85,B 0,C 180,E1 4915.655,E2 4915.655} C_VEL
LIN {X 0,Y 96.953,Z 592.595,A -85,B 0,C 180,E1 4910.677,E2 4910.677} C_VEL
LIN {X 0,Y 99.907,Z 574.154,A -85,B 0,C 180,E1 4906.792,E2 4906.792} C_VEL
LIN {X 0,Y 102.054,Z 554.928,A -85,B 0,C 180,E1 4903.928,E2 4903.928} C_VEL
LIN {X 0,Y 116.929,Z 432.946,A -85,B 0,C 180,E1 4890.804,E2 4890.804} C_VEL
LIN {X 0,Y 114.528,Z 426.555,A -85,B 0,C 180,E1 4889.533,E2 4889.533} C_VEL
LIN {X 0,Y 111.172,Z 420.273,A -85,B 0,C 180,E1 4887.965,E2 4887.965} C_VEL
LIN {X 0,Y 98.653,Z 404.685,A -85,B 0,C 180,E1 4882.411,E2 4882.411} C_VEL
LIN {X 0,Y 96.356,Z 400.215,A -85,B 0,C 180,E1 4880.981,E2 4880.981} C_VEL
LIN {X 0,Y 94.04,Z 394.458,A -85,B 0,C 180,E1 4879.253,E2 4879.253} C_VEL
LIN {X 0,Y 91.746,Z 385.019,A -85,B 0,C 180,E1 4871.959,E2 4871.959} C_VEL
LIN {X 0,Y 89.593,Z 376.768,A -85,B 0,C 180,E1 4864.49,E2 4864.49} C_VEL
LIN {X 0,Y 87.709,Z 370.167,A -85,B 0,C 180,E1 4857.396,E2 4857.396} C_VEL
LIN {X 0,Y 85.864,Z 364.502,A -85,B 0,C 180,E1 4849.95,E2 4849.95} C_VEL
LIN {X 0,Y 84.577,Z 360.992,A -85,B 0,C 180,E1 4844.233,E2 4844.233} C_VEL
LIN {X 0,Y 83.61,Z 358.189,A -85,B 0,C 180,E1 4838.855,E2 4838.855} C_VEL
LIN {X 0,Y 82.338,Z 354.762,A -85,B 0,C 180,E1 4830.153,E2 4830.153} C_VEL
LIN {X 0,Y 81.1,Z 352.301,A -85,B 0,C 180,E1 4818.275,E2 4818.275} C_VEL
LIN {X 0,Y 80.946,Z 351.626,A -85,B 0,C 180,E1 4809.957,E2 4809.957} C_VEL
LIN {X 0,Y 81.028,Z 352.201,A -85,B 0,C 180,E1 4801.653,E2 4801.653} C_VEL
LIN {X 0,Y 81.847,Z 354.117,A -85,B 0,C 180,E1 4791.493,E2 4791.493} C_VEL
LIN {X 0,Y 82.514,Z 355.432,A -85,B 0,C 180,E1 4786.847,E2 4786.847} C_VEL
LIN {X 0,Y 83.826,Z 359.076,A -85,B 0,C 180,E1 4778.185,E2 4778.185} C_VEL
LIN {X 0,Y 85.011,Z 362.657,A -85,B 0,C 180,E1 4771.743,E2 4771.743} C_VEL
LIN {X 0,Y 86.557,Z 367.435,A -85,B 0,C 180,E1 4764.693,E2 4764.693} C_VEL
LIN {X 0,Y 88.366,Z 373.984,A -85,B 0,C 180,E1 4756.916,E2 4756.916} C_VEL
LIN {X 0,Y 90.156,Z 381.829,A -85,B 0,C 180,E1 4749.208,E2 4749.208} C_VEL
LIN {X 0,Y 91.916,Z 390.688,A -85,B 0,C 180,E1 4741.756,E2 4741.756} C_VEL
LIN {X 0,Y 93.306,Z 398.114,A -85,B 0,C 180,E1 4736.407,E2 4736.407} C_VEL
LIN {X 0,Y 97.424,Z 411.025,A -85,B 0,C 180,E1 4732.95,E2 4732.95} C_VEL
LIN {X 0,Y 96.517,Z 450.243,A -85,B 0,C 180,E1 4727.019,E2 4727.019} C_VEL
LIN {X 0,Y 95.836,Z 456.842,A -85,B 0,C 180,E1 4726.138,E2 4726.138} C_VEL
LIN {X 0,Y 83.716,Z 552.238,A -85,B 0,C 180,E1 4712.04,E2 4712.04} C_VEL
LIN {X 0,Y 81.244,Z 571.701,A -85,B 0,C 180,E1 4707.512,E2 4707.512} C_VEL
LIN {X 0,Y 78.829,Z 590.338,A -85,B 0,C 180,E1 4701.57,E2 4701.57} C_VEL
LIN {X 0,Y 76.868,Z 608.451,A -85,B 0,C 180,E1 4693.913,E2 4693.913} C_VEL
LIN {X 0,Y 76.046,Z 624.441,A -85,B 0,C 180,E1 4685.27,E2 4685.27} C_VEL
LIN {X 0,Y 76.702,Z 639.218,A -85,B 0,C 180,E1 4675.504,E2 4675.504} C_VEL
LIN {X 0,Y 79.302,Z 652.171,A -85,B 0,C 180,E1 4665.384,E2 4665.384} C_VEL
LIN {X 0,Y 84.806,Z 664.474,A -85,B 0,C 180,E1 4654.875,E2 4654.875} C_VEL
LIN {X 0,Y 93.526,Z 675.231,A -85,B 0,C 180,E1 4645.476,E2 4645.476} C_VEL
LIN {X 0,Y 98.672,Z 679.81,A -85,B 0,C 180,E1 4641.523,E2 4641.523} C_VEL
LIN {X 0,Y 86.551,Z 677.663,A -85,B 0,C 180,E1 4626.927,E2 4626.927} C_VEL
LIN {X 0,Y 82.494,Z 673.932,A -85,B 0,C 180,E1 4609.107,E2 4609.107} C_VEL
LIN {X 0,Y 85.377,Z 669.398,A -85,B 0,C 180,E1 4594.984,E2 4594.984} C_VEL
LIN {X 0,Y 82.795,Z 660.501,A -85,B 0,C 180,E1 4586.544,E2 4586.544} C_VEL
LIN {X 0,Y 81.592,Z 648.805,A -85,B 0,C 180,E1 4577.262,E2 4577.262} C_VEL
LIN {X 0,Y 82.127,Z 635.385,A -85,B 0,C 180,E1 4568.584,E2 4568.584} C_VEL
LIN {X 0,Y 84.056,Z 620.259,A -85,B 0,C 180,E1 4560.817,E2 4560.817} C_VEL
LIN {X 0,Y 86.812,Z 603.975,A -85,B 0,C 180,E1 4554.441,E2 4554.441} C_VEL
LIN {X 0,Y 89.843,Z 586.725,A -85,B 0,C 180,E1 4549.386,E2 4549.386} C_VEL
LIN {X 0,Y 92.509,Z 569.25,A -85,B 0,C 180,E1 4545.674,E2 4545.674} C_VEL
LIN {X 0,Y 95.594,Z 540.441,A -85,B 0,C 180,E1 4541.462,E2 4541.462} C_VEL
LIN {X 0,Y 109.351,Z 434.549,A -85,B 0,C 180,E1 4529.377,E2 4529.377} C_VEL
LIN {X 0,Y 98.339,Z 405.162,A -85,B 0,C 180,E1 4522.386,E2 4522.386} C_VEL
LIN {X 0,Y 96.356,Z 400.215,A -85,B 0,C 180,E1 4520.981,E2 4520.981} C_VEL
LIN {X 0,Y 93.911,Z 395.223,A -85,B 0,C 180,E1 4518.831,E2 4518.831} C_VEL
LIN {X 0,Y 90.268,Z 390.208,A -85,B 0,C 180,E1 4514.85,E2 4514.85} C_VEL
LIN {X 0,Y 83.318,Z 382.101,A -85,B 0,C 180,E1 4504.987,E2 4504.987} C_VEL
LIN {X 0,Y 82.869,Z 380.921,A -85,B 0,C 180,E1 4503.668,E2 4503.668} C_VEL
LIN {X 0,Y 81.155,Z 374.474,A -85,B 0,C 180,E1 4496.239,E2 4496.239} C_VEL
LIN {X 0,Y 79.535,Z 369.12,A -85,B 0,C 180,E1 4488.656,E2 4488.656} C_VEL
LIN {X 0,Y 78.43,Z 365.856,A -85,B 0,C 180,E1 4482.945,E2 4482.945} C_VEL
LIN {X 0,Y 77.66,Z 363.439,A -85,B 0,C 180,E1 4477.954,E2 4477.954} C_VEL
LIN {X 0,Y 76.595,Z 360.295,A -85,B 0,C 180,E1 4469.409,E2 4469.409} C_VEL
LIN {X 0,Y 75.535,Z 357.992,A -85,B 0,C 180,E1 4457.555,E2 4457.555} C_VEL
LIN {X 0,Y 75.436,Z 357.426,A -85,B 0,C 180,E1 4448.525,E2 4448.525} C_VEL
LIN {X 0,Y 75.57,Z 358.318,A -85,B 0,C 180,E1 4439.188,E2 4439.188} C_VEL
LIN {X 0,Y 76.682,Z 360.591,A -85,B 0,C 180,E1 4428.23,E2 4428.23} C_VEL
LIN {X 0,Y 77.815,Z 364.296,A -85,B 0,C 180,E1 4418.864,E2 4418.864} C_VEL
LIN {X 0,Y 78.876,Z 367.82,A -85,B 0,C 180,E1 4412.174,E2 4412.174} C_VEL
LIN {X 0,Y 80.223,Z 372.483,A -85,B 0,C 180,E1 4404.989,E2 4404.989} C_VEL
LIN {X 0,Y 81.747,Z 378.641,A -85,B 0,C 180,E1 4397.276,E2 4397.276} C_VEL
LIN {X 0,Y 83.325,Z 386.277,A -85,B 0,C 180,E1 4389.352,E2 4389.352} C_VEL
LIN {X 0,Y 84.824,Z 394.739,A -85,B 0,C 180,E1 4381.863,E2 4381.863} C_VEL
LIN {X 0,Y 85.45,Z 398.023,A -85,B 0,C 180,E1 4379.446,E2 4379.446} C_VEL
LIN {X 0,Y 90.218,Z 412.784,A -85,B 0,C 180,E1 4374.978,E2 4374.978} C_VEL
LIN {X 0,Y 88.815,Z 453.908,A -85,B 0,C 180,E1 4368.305,E2 4368.305} C_VEL
LIN {X 0,Y 75.71,Z 552.285,A -85,B 0,C 180,E1 4352.545,E2 4352.545} C_VEL
LIN {X 0,Y 73.226,Z 571.401,A -85,B 0,C 180,E1 4347.649,E2 4347.649} C_VEL
LIN {X 0,Y 70.699,Z 590.962,A -85,B 0,C 180,E1 4340.692,E2 4340.692} C_VEL
LIN {X 0,Y 68.912,Z 608.938,A -85,B 0,C 180,E1 4332.132,E2 4332.132} C_VEL
LIN {X 0,Y 68.45,Z 624.824,A -85,B 0,C 180,E1 4322.5,E2 4322.5} C_VEL
LIN {X 0,Y 69.706,Z 639.506,A -85,B 0,C 180,E1 4311.741,E2 4311.741} C_VEL
LIN {X 0,Y 73.153,Z 652.432,A -85,B 0,C 180,E1 4300.839,E2 4300.839} C_VEL
LIN {X 0,Y 80.328,Z 665.429,A -85,B 0,C 180,E1 4289.303,E2 4289.303} C_VEL
LIN {X 0,Y 89.43,Z 675.328,A -85,B 0,C 180,E1 4280.773,E2 4280.773} C_VEL
LIN {X 0,Y 78.407,Z 672.426,A -85,B 0,C 180,E1 4264.138,E2 4264.138} C_VEL
LIN {X 0,Y 76.321,Z 668.251,A -85,B 0,C 180,E1 4245.975,E2 4245.975} C_VEL
LIN {X 0,Y 78.467,Z 665.088,A -85,B 0,C 180,E1 4236.247,E2 4236.247} C_VEL
LIN {X 0,Y 75.604,Z 655.548,A -85,B 0,C 180,E1 4226.973,E2 4226.973} C_VEL
LIN {X 0,Y 74.354,Z 643.701,A -85,B 0,C 180,E1 4217.187,E2 4217.187} C_VEL
LIN {X 0,Y 74.915,Z 630.149,A -85,B 0,C 180,E1 4208.062,E2 4208.062} C_VEL
LIN {X 0,Y 77.005,Z 614.142,A -85,B 0,C 180,E1 4199.583,E2 4199.583} C_VEL
LIN {X 0,Y 79.594,Z 598.886,A -85,B 0,C 180,E1 4193.418,E2 4193.418} C_VEL
LIN {X 0,Y 82.814,Z 580.379,A -85,B 0,C 180,E1 4187.934,E2 4187.934} C_VEL
LIN {X 0,Y 85.233,Z 562.965,A -85,B 0,C 180,E1 4184.227,E2 4184.227} C_VEL
LIN {X 0,Y 101.448,Z 439.192,A -85,B 0,C 180,E1 4168.173,E2 4168.173} C_VEL
LIN {X 0,Y 101.678,Z 435.892,A -85,B 0,C 180,E1 4167.767,E2 4167.767} C_VEL
LIN {X 0,Y 91.37,Z 407.916,A -85,B 0,C 180,E1 4160.507,E2 4160.507} C_VEL
LIN {X 0,Y 86.078,Z 394.444,A -85,B 0,C 180,E1 4156.024,E2 4156.024} C_VEL
LIN {X 0,Y 84.004,Z 385.514,A -85,B 0,C 180,E1 4148.221,E2 4148.221} C_VEL
LIN {X 0,Y 82.869,Z 380.921,A -85,B 0,C 180,E1 4143.668,E2 4143.668} C_VEL
LIN {X 0,Y 81.241,Z 377.91,A -85,B 0,C 180,E1 4139.696,E2 4139.696} C_VEL
LIN {X 0,Y 77.978,Z 375.148,A -85,B 0,C 180,E1 4134.028,E2 4134.028} C_VEL
LIN {X 0,Y 72.415,Z 370.744,A -85,B 0,C 180,E1 4121.597,E2 4121.597} C_VEL
LIN {X 0,Y 72.103,Z 369.759,A -85,B 0,C 180,E1 4119.478,E2 4119.478} C_VEL
LIN {X 0,Y 70.944,Z 365.956,A -85,B 0,C 180,E1 4109.271,E2 4109.271} C_VEL
LIN {X 0,Y 69.98,Z 363.686,A -85,B 0,C 180,E1 4096.717,E2 4096.717} C_VEL
LIN {X 0,Y 69.922,Z 363.244,A -85,B 0,C 180,E1 4087.935,E2 4087.935} C_VEL
LIN {X 0,Y 70.056,Z 364.305,A -85,B 0,C 180,E1 4077.791,E2 4077.791} C_VEL
LIN {X 0,Y 70.899,Z 366.082,A -85,B 0,C 180,E1 4068.92,E2 4068.92} C_VEL
LIN {X 0,Y 71.829,Z 369.546,A -85,B 0,C 180,E1 4059.61,E2 4059.61} C_VEL
LIN {X 0,Y 72.805,Z 373.165,A -85,B 0,C 180,E1 4052.355,E2 4052.355} C_VEL
LIN {X 0,Y 74.037,Z 378.035,A -85,B 0,C 180,E1 4044.57,E2 4044.57} C_VEL
LIN {X 0,Y 75.393,Z 384.568,A -85,B 0,C 180,E1 4036.183,E2 4036.183} C_VEL
LIN {X 0,Y 76.765,Z 392.478,A -85,B 0,C 180,E1 4027.801,E2 4027.801} C_VEL
LIN {X 0,Y 77.609,Z 397.73,A -85,B 0,C 180,E1 4023.088,E2 4023.088} C_VEL
LIN {X 0,Y 82.795,Z 413.476,A -85,B 0,C 180,E1 4017.59,E2 4017.59} C_VEL
LIN {X 0,Y 82.981,Z 415.868,A -85,B 0,C 180,E1 4017.057,E2 4017.057} C_VEL
LIN {X 0,Y 81.358,Z 454.109,A -85,B 0,C 180,E1 4010.326,E2 4010.326} C_VEL
LIN {X 0,Y 67.613,Z 552.97,A -85,B 0,C 180,E1 3992.904,E2 3992.904} C_VEL
LIN {X 0,Y 64.928,Z 573.08,A -85,B 0,C 180,E1 3987.004,E2 3987.004} C_VEL
LIN {X 0,Y 62.51,Z 592.288,A -85,B 0,C 180,E1 3979.127,E2 3979.127} C_VEL
LIN {X 0,Y 60.994,Z 610.739,A -85,B 0,C 180,E1 3968.945,E2 3968.945} C_VEL
LIN {X 0,Y 61.161,Z 626.249,A -85,B 0,C 180,E1 3958.113,E2 3958.113} C_VEL
LIN {X 0,Y 63.332,Z 640.624,A -85,B 0,C 180,E1 3946.288,E2 3946.288} C_VEL
LIN {X 0,Y 67.98,Z 653.357,A -85,B 0,C 180,E1 3934.739,E2 3934.739} C_VEL
LIN {X 0,Y 76.718,Z 666.228,A -85,B 0,C 180,E1 3923.153,E2 3923.153} C_VEL
LIN {X 0,Y 80.445,Z 670.243,A -85,B 0,C 180,E1 3919.612,E2 3919.612} C_VEL
LIN {X 0,Y 70.842,Z 666.594,A -85,B 0,C 180,E1 3900.545,E2 3900.545} C_VEL
LIN {X 0,Y 71.041,Z 661.617,A -85,B 0,C 180,E1 3880.549,E2 3880.549} C_VEL
LIN {X 0,Y 71.659,Z 660.559,A -85,B 0,C 180,E1 3877.761,E2 3877.761} C_VEL
LIN {X 0,Y 68.466,Z 650.319,A -85,B 0,C 180,E1 3867.495,E2 3867.495} C_VEL
LIN {X 0,Y 67.187,Z 638.215,A -85,B 0,C 180,E1 3857.108,E2 3857.108} C_VEL
LIN {X 0,Y 67.757,Z 624.596,A -85,B 0,C 180,E1 3847.446,E2 3847.446} C_VEL
LIN {X 0,Y 69.763,Z 609.282,A -85,B 0,C 180,E1 3838.946,E2 3838.946} C_VEL
LIN {X 0,Y 72.681,Z 592.026,A -85,B 0,C 180,E1 3831.761,E2 3831.761} C_VEL
LIN {X 0,Y 75.735,Z 574.02,A -85,B 0,C 180,E1 3826.393,E2 3826.393} C_VEL
LIN {X 0,Y 78.079,Z 555.173,A -85,B 0,C 180,E1 3822.441,E2 3822.441} C_VEL
LIN {X 0,Y 94.171,Z 437.664,A -85,B 0,C 180,E1 3806.094,E2 3806.094} C_VEL
LIN {X 0,Y 84.507,Z 410.726,A -85,B 0,C 180,E1 3798.416,E2 3798.416} C_VEL
LIN {X 0,Y 78.274,Z 394.8,A -85,B 0,C 180,E1 3792.552,E2 3792.552} C_VEL
LIN {X 0,Y 76.389,Z 386.027,A -85,B 0,C 180,E1 3783.763,E2 3783.763} C_VEL
LIN {X 0,Y 74.748,Z 379.131,A -85,B 0,C 180,E1 3775.408,E2 3775.408} C_VEL
LIN {X 0,Y 73.299,Z 373.876,A -85,B 0,C 180,E1 3767.405,E2 3767.405} C_VEL
LIN {X 0,Y 72.103,Z 369.759,A -85,B 0,C 180,E1 3759.478,E2 3759.478} C_VEL
LIN {X 0,Y 71.184,Z 368.174,A -85,B 0,C 180,E1 3754.861,E2 3754.861} C_VEL
LIN {X 0,Y 69.276,Z 367.641,A -85,B 0,C 180,E1 3749.174,E2 3749.174} C_VEL
LIN {X 0,Y 65.738,Z 368.488,A -85,B 0,C 180,E1 3738.834,E2 3738.834} C_VEL
LIN {X 0,Y 64.427,Z 369.037,A -85,B 0,C 180,E1 3729.636,E2 3729.636} C_VEL
LIN {X 0,Y 64.416,Z 369.665,A -85,B 0,C 180,E1 3720.804,E2 3720.804} C_VEL
LIN {X 0,Y 65.168,Z 371.619,A -85,B 0,C 180,E1 3709.72,E2 3709.72} C_VEL
LIN {X 0,Y 65.878,Z 374.816,A -85,B 0,C 180,E1 3700.487,E2 3700.487} C_VEL
LIN {X 0,Y 66.758,Z 378.518,A -85,B 0,C 180,E1 3692.569,E2 3692.569} C_VEL
LIN {X 0,Y 67.78,Z 383.638,A -85,B 0,C 180,E1 3684.067,E2 3684.067} C_VEL
LIN {X 0,Y 68.844,Z 389.954,A -85,B 0,C 180,E1 3675.699,E2 3675.699} C_VEL
LIN {X 0,Y 69.967,Z 397.566,A -85,B 0,C 180,E1 3667.464,E2 3667.464} C_VEL
LIN {X 0,Y 74.797,Z 412.107,A -85,B 0,C 180,E1 3661.391,E2 3661.391} C_VEL
LIN {X 0,Y 75.965,Z 417.068,A -85,B 0,C 180,E1 3659.761,E2 3659.761} C_VEL
LIN {X 0,Y 73.996,Z 454.128,A -85,B 0,C 180,E1 3652.686,E2 3652.686} C_VEL
LIN {X 0,Y 59.552,Z 553.264,A -85,B 0,C 180,E1 3633.34,E2 3633.34} C_VEL
LIN {X 0,Y 56.827,Z 573.284,A -85,B 0,C 180,E1 3626.641,E2 3626.641} C_VEL
LIN {X 0,Y 54.505,Z 592.414,A -85,B 0,C 180,E1 3617.602,E2 3617.602} C_VEL
LIN {X 0,Y 53.368,Z 610.001,A -85,B 0,C 180,E1 3606.439,E2 3606.439} C_VEL
LIN {X 0,Y 54.008,Z 625.042,A -85,B 0,C 180,E1 3594.674,E2 3594.674} C_VEL
LIN {X 0,Y 56.841,Z 639.012,A -85,B 0,C 180,E1 3582.057,E2 3582.057} C_VEL
LIN {X 0,Y 62.699,Z 652.412,A -85,B 0,C 180,E1 3569.301,E2 3569.301} C_VEL
LIN {X 0,Y 71.936,Z 664.732,A -85,B 0,C 180,E1 3558.198,E2 3558.198} C_VEL
LIN {X 0,Y 64.062,Z 660.454,A -85,B 0,C 180,E1 3536.919,E2 3536.919} C_VEL
LIN {X 0,Y 65.102,Z 656.129,A -85,B 0,C 180,E1 3519.956,E2 3519.956} C_VEL
LIN {X 0,Y 61.586,Z 645.74,A -85,B 0,C 180,E1 3509.077,E2 3509.077} C_VEL
LIN {X 0,Y 60.089,Z 632.992,A -85,B 0,C 180,E1 3497.515,E2 3497.515} C_VEL
LIN {X 0,Y 60.673,Z 618.611,A -85,B 0,C 180,E1 3486.71,E2 3486.71} C_VEL
LIN {X 0,Y 62.748,Z 603.002,A -85,B 0,C 180,E1 3477.644,E2 3477.644} C_VEL
LIN {X 0,Y 65.662,Z 585.765,A -85,B 0,C 180,E1 3470.251,E2 3470.251} C_VEL
LIN {X 0,Y 68.475,Z 568.427,A -85,B 0,C 180,E1 3464.922,E2 3464.922} C_VEL
LIN {X 0,Y 71.36,Z 543.683,A -85,B 0,C 180,E1 3459.796,E2 3459.796} C_VEL
LIN {X 0,Y 86.615,Z 439.112,A -85,B 0,C 180,E1 3444.138,E2 3444.138} C_VEL
LIN {X 0,Y 77.476,Z 412.889,A -85,B 0,C 180,E1 3435.831,E2 3435.831} C_VEL
LIN {X 0,Y 71.616,Z 397.656,A -85,B 0,C 180,E1 3429.453,E2 3429.453} C_VEL
LIN {X 0,Y 70.553,Z 394.993,A -85,B 0,C 180,E1 3428.159,E2 3428.159} C_VEL
LIN {X 0,Y 69.056,Z 387.245,A -85,B 0,C 180,E1 3419.182,E2 3419.182} C_VEL
LIN {X 0,Y 67.747,Z 381.281,A -85,B 0,C 180,E1 3410.669,E2 3410.669} C_VEL
LIN {X 0,Y 66.502,Z 376.402,A -85,B 0,C 180,E1 3401.608,E2 3401.608} C_VEL
LIN {X 0,Y 65.812,Z 373.915,A -85,B 0,C 180,E1 3395.705,E2 3395.705} C_VEL
LIN {X 0,Y 65.105,Z 371.326,A -85,B 0,C 180,E1 3387.501,E2 3387.501} C_VEL
LIN {X 0,Y 64.455,Z 369.383,A -85,B 0,C 180,E1 3375.517,E2 3375.517} C_VEL
LIN {X 0,Y 64.427,Z 369.037,A -85,B 0,C 180,E1 3369.636,E2 3369.636} C_VEL
LIN {X 0,Y 64.04,Z 369.696,A -85,B 0,C 180,E1 3364.281,E2 3364.281} C_VEL
LIN {X 0,Y 62.855,Z 371.84,A -85,B 0,C 180,E1 3358.121,E2 3358.121} C_VEL
LIN {X 0,Y 60.39,Z 377.622,A -85,B 0,C 180,E1 3346.586,E2 3346.586} C_VEL
LIN {X 0,Y 60.187,Z 381.306,A -85,B 0,C 180,E1 3338.387,E2 3338.387} C_VEL
LIN {X 0,Y 60.905,Z 385.375,A -85,B 0,C 180,E1 3329.993,E2 3329.993} C_VEL
LIN {X 0,Y 61.707,Z 391.236,A -85,B 0,C 180,E1 3320.668,E2 3320.668} C_VEL
LIN {X 0,Y 62.536,Z 397.533,A -85,B 0,C 180,E1 3312.788,E2 3312.788} C_VEL
LIN {X 0,Y 66.811,Z 410.362,A -85,B 0,C 180,E1 3306.219,E2 3306.219} C_VEL
LIN {X 0,Y 69.036,Z 418.745,A -85,B 0,C 180,E1 3302.82,E2 3302.82} C_VEL
LIN {X 0,Y 66.711,Z 454.221,A -85,B 0,C 180,E1 3295.45,E2 3295.45} C_VEL
LIN {X 0,Y 51.506,Z 553.353,A -85,B 0,C 180,E1 3273.818,E2 3273.818} C_VEL
LIN {X 0,Y 48.808,Z 572.897,A -85,B 0,C 180,E1 3266.264,E2 3266.264} C_VEL
LIN {X 0,Y 46.683,Z 591.298,A -85,B 0,C 180,E1 3256.148,E2 3256.148} C_VEL
LIN {X 0,Y 45.904,Z 608.326,A -85,B 0,C 180,E1 3243.729,E2 3243.729} C_VEL
LIN {X 0,Y 47.177,Z 623.552,A -85,B 0,C 180,E1 3230.221,E2 3230.221} C_VEL
LIN {X 0,Y 50.783,Z 637.229,A -85,B 0,C 180,E1 3216.793,E2 3216.793} C_VEL
LIN {X 0,Y 57.534,Z 650.464,A -85,B 0,C 180,E1 3203.764,E2 3203.764} C_VEL
LIN {X 0,Y 63.784,Z 658.664,A -85,B 0,C 180,E1 3196.153,E2 3196.153} C_VEL
LIN {X 0,Y 57.924,Z 653.841,A -85,B 0,C 180,E1 3172.327,E2 3172.327} C_VEL
LIN {X 0,Y 58.713,Z 651.362,A -85,B 0,C 180,E1 3162.548,E2 3162.548} C_VEL
LIN {X 0,Y 54.72,Z 640.373,A -85,B 0,C 180,E1 3150.531,E2 3150.531} C_VEL
LIN {X 0,Y 53.047,Z 627.479,A -85,B 0,C 180,E1 3138.042,E2 3138.042} C_VEL
LIN {X 0,Y 53.62,Z 612.535,A -85,B 0,C 180,E1 3126.058,E2 3126.058} C_VEL
LIN {X 0,Y 55.748,Z 596.574,A -85,B 0,C 180,E1 3116.23,E2 3116.23} C_VEL
LIN {X 0,Y 58.725,Z 578.918,A -85,B 0,C 180,E1 3108.403,E2 3108.403} C_VEL
LIN {X 0,Y 61.231,Z 562.18,A -85,B 0,C 180,E1 3103.159,E2 3103.159} C_VEL
LIN {X 0,Y 77.345,Z 451.582,A -85,B 0,C 180,E1 3083.404,E2 3083.404} C_VEL
LIN {X 0,Y 79.107,Z 440.511,A -85,B 0,C 180,E1 3081.903,E2 3081.903} C_VEL
LIN {X 0,Y 70.588,Z 415.208,A -85,B 0,C 180,E1 3072.902,E2 3072.902} C_VEL
LIN {X 0,Y 65.25,Z 400.748,A -85,B 0,C 180,E1 3066.06,E2 3066.06} C_VEL
LIN {X 0,Y 63.015,Z 395.156,A -85,B 0,C 180,E1 3062.741,E2 3062.741} C_VEL
LIN {X 0,Y 61.901,Z 388.504,A -85,B 0,C 180,E1 3053.521,E2 3053.521} C_VEL
LIN {X 0,Y 60.912,Z 383.535,A -85,B 0,C 180,E1 3044.788,E2 3044.788} C_VEL
LIN {X 0,Y 60.068,Z 379.504,A -85,B 0,C 180,E1 3035.425,E2 3035.425} C_VEL
LIN {X 0,Y 59.495,Z 377.017,A -85,B 0,C 180,E1 3027.157,E2 3027.157} C_VEL
LIN {X 0,Y 58.945,Z 375.128,A -85,B 0,C 180,E1 3014.588,E2 3014.588} C_VEL
LIN {X 0,Y 58.925,Z 374.963,A -85,B 0,C 180,E1 3006.424,E2 3006.424} C_VEL
LIN {X 0,Y 59.083,Z 376.334,A -85,B 0,C 180,E1 2995.021,E2 2995.021} C_VEL
LIN {X 0,Y 59.432,Z 377.461,A -85,B 0,C 180,E1 2989.634,E2 2989.634} C_VEL
LIN {X 0,Y 59.919,Z 380.05,A -85,B 0,C 180,E1 2981.544,E2 2981.544} C_VEL
LIN {X 0,Y 60.187,Z 381.306,A -85,B 0,C 180,E1 2978.387,E2 2978.387} C_VEL
LIN {X 0,Y 59.986,Z 383.391,A -85,B 0,C 180,E1 2974.741,E2 2974.741} C_VEL
LIN {X 0,Y 58.213,Z 387.72,A -85,B 0,C 180,E1 2970.073,E2 2970.073} C_VEL
LIN {X 0,Y 55.324,Z 394.63,A -85,B 0,C 180,E1 2963.107,E2 2963.107} C_VEL
LIN {X 0,Y 55.133,Z 396.518,A -85,B 0,C 180,E1 2960.549,E2 2960.549} C_VEL
LIN {X 0,Y 58.34,Z 406.107,A -85,B 0,C 180,E1 2953.731,E2 2953.731} C_VEL
LIN {X 0,Y 62.199,Z 419.831,A -85,B 0,C 180,E1 2946.661,E2 2946.661} C_VEL
LIN {X 0,Y 59.592,Z 454.1,A -85,B 0,C 180,E1 2938.808,E2 2938.808} C_VEL
LIN {X 0,Y 43.493,Z 553.136,A -85,B 0,C 180,E1 2914.405,E2 2914.405} C_VEL
LIN {X 0,Y 40.736,Z 572.964,A -85,B 0,C 180,E1 2905.284,E2 2905.284} C_VEL
LIN {X 0,Y 38.841,Z 591.469,A -85,B 0,C 180,E1 2892.924,E2 2892.924} C_VEL
LIN {X 0,Y 38.718,Z 607.974,A -85,B 0,C 180,E1 2878.499,E2 2878.499} C_VEL
LIN {X 0,Y 41.078,Z 623.148,A -85,B 0,C 180,E1 2862.997,E2 2862.997} C_VEL
LIN {X 0,Y 46.073,Z 636.756,A -85,B 0,C 180,E1 2848.591,E2 2848.591} C_VEL
LIN {X 0,Y 55.079,Z 650.877,A -85,B 0,C 180,E1 2834.91,E2 2834.91} C_VEL
LIN {X 0,Y 56.182,Z 652.222,A -85,B 0,C 180,E1 2833.611,E2 2833.611} C_VEL
LIN {X 0,Y 52.619,Z 646.706,A -85,B 0,C 180,E1 2806.569,E2 2806.569} C_VEL
LIN {X 0,Y 52.425,Z 646.126,A -85,B 0,C 180,E1 2805.495,E2 2805.495} C_VEL
LIN {X 0,Y 47.978,Z 634.65,A -85,B 0,C 180,E1 2792.398,E2 2792.398} C_VEL
LIN {X 0,Y 46.07,Z 621.625,A -85,B 0,C 180,E1 2778.746,E2 2778.746} C_VEL
LIN {X 0,Y 46.543,Z 606.898,A -85,B 0,C 180,E1 2765.921,E2 2765.921} C_VEL
LIN {X 0,Y 48.708,Z 590.385,A -85,B 0,C 180,E1 2754.928,E2 2754.928} C_VEL
LIN {X 0,Y 51.545,Z 573.352,A -85,B 0,C 180,E1 2746.873,E2 2746.873} C_VEL
LIN {X 0,Y 53.974,Z 555.635,A -85,B 0,C 180,E1 2741.149,E2 2741.149} C_VEL
LIN {X 0,Y 71.699,Z 442.034,A -85,B 0,C 180,E1 2719.353,E2 2719.353} C_VEL
LIN {X 0,Y 63.929,Z 417.743,A -85,B 0,C 180,E1 2709.595,E2 2709.595} C_VEL
LIN {X 0,Y 59.015,Z 403.606,A -85,B 0,C 180,E1 2701.861,E2 2701.861} C_VEL
LIN {X 0,Y 55.7,Z 395.056,A -85,B 0,C 180,E1 2695.382,E2 2695.382} C_VEL
LIN {X 0,Y 55.007,Z 389.928,A -85,B 0,C 180,E1 2686.347,E2 2686.347} C_VEL
LIN {X 0,Y 54.366,Z 385.965,A -85,B 0,C 180,E1 2677.297,E2 2677.297} C_VEL
LIN {X 0,Y 53.914,Z 382.76,A -85,B 0,C 180,E1 2667.072,E2 2667.072} C_VEL
LIN {X 0,Y 53.451,Z 380.898,A -85,B 0,C 180,E1 2653.787,E2 2653.787} C_VEL
LIN {X 0,Y 53.437,Z 380.804,A -85,B 0,C 180,E1 2646.458,E2 2646.458} C_VEL
LIN {X 0,Y 53.58,Z 382.29,A -85,B 0,C 180,E1 2633.921,E2 2633.921} C_VEL
LIN {X 0,Y 53.985,Z 384.701,A -85,B 0,C 180,E1 2624.471,E2 2624.471} C_VEL
LIN {X 0,Y 54.413,Z 388.309,A -85,B 0,C 180,E1 2615.264,E2 2615.264} C_VEL
LIN {X 0,Y 54.898,Z 393.25,A -85,B 0,C 180,E1 2605.814,E2 2605.814} C_VEL
LIN {X 0,Y 55.133,Z 396.518,A -85,B 0,C 180,E1 2600.549,E2 2600.549} C_VEL
LIN {X 0,Y 57.278,Z 401.294,A -85,B 0,C 180,E1 2596.294,E2 2596.294} C_VEL
LIN {X 0,Y 58.308,Z 406.264,A -85,B 0,C 180,E1 2593.755,E2 2593.755} C_VEL
LIN {X 0,Y 58.274,Z 412.892,A -85,B 0,C 180,E1 2591.769,E2 2591.769} C_VEL
LIN {X 0,Y 56.797,Z 421.131,A -85,B 0,C 180,E1 2590.528,E2 2590.528} C_VEL
LIN {X 0,Y 54.802,Z 430.507,A -85,B 0,C 180,E1 2588.864,E2 2588.864} C_VEL
LIN {X 0,Y 52.634,Z 454.096,A -85,B 0,C 180,E1 2582.912,E2 2582.912} C_VEL
LIN {X 0,Y 35.518,Z 552.596,A -85,B 0,C 180,E1 2555.156,E2 2555.156} C_VEL
LIN {X 0,Y 32.843,Z 571.775,A -85,B 0,C 180,E1 2544.45,E2 2544.45} C_VEL
LIN {X 0,Y 31.257,Z 590.282,A -85,B 0,C 180,E1 2529.177,E2 2529.177} C_VEL
LIN {X 0,Y 32.06,Z 607.345,A -85,B 0,C 180,E1 2511.003,E2 2511.003} C_VEL
LIN {X 0,Y 35.649,Z 621.954,A -85,B 0,C 180,E1 2494.207,E2 2494.207} C_VEL
LIN {X 0,Y 41.892,Z 635.103,A -85,B 0,C 180,E1 2479.854,E2 2479.854} C_VEL
LIN {X 0,Y 49.082,Z 645.328,A -85,B 0,C 180,E1 2470.164,E2 2470.164} C_VEL
LIN {X 0,Y 46.933,Z 641.531,A -85,B 0,C 180,E1 2450.339,E2 2450.339} C_VEL
LIN {X 0,Y 41.697,Z 629.702,A -85,B 0,C 180,E1 2436.205,E2 2436.205} C_VEL
LIN {X 0,Y 39.237,Z 615.999,A -85,B 0,C 180,E1 2420.477,E2 2420.477} C_VEL
LIN {X 0,Y 39.533,Z 600.723,A -85,B 0,C 180,E1 2405.623,E2 2405.623} C_VEL
LIN {X 0,Y 41.744,Z 583.677,A -85,B 0,C 180,E1 2393.229,E2 2393.229} C_VEL
LIN {X 0,Y 44.519,Z 566.504,A -85,B 0,C 180,E1 2384.643,E2 2384.643} C_VEL
LIN {X 0,Y 47.606,Z 542.124,A -85,B 0,C 180,E1 2376.752,E2 2376.752} C_VEL
LIN {X 0,Y 64.364,Z 443.45,A -85,B 0,C 180,E1 2356.308,E2 2356.308} C_VEL
LIN {X 0,Y 57.611,Z 420.96,A -85,B 0,C 180,E1 2345.991,E2 2345.991} C_VEL
LIN {X 0,Y 53.433,Z 407.736,A -85,B 0,C 180,E1 2337.736,E2 2337.736} C_VEL
LIN {X 0,Y 50.2,Z 398.967,A -85,B 0,C 180,E1 2330.125,E2 2330.125} C_VEL
LIN {X 0,Y 48.833,Z 395.271,A -85,B 0,C 180,E1 2325.794,E2 2325.794} C_VEL
LIN {X 0,Y 48.458,Z 391.162,A -85,B 0,C 180,E1 2315.647,E2 2315.647} C_VEL
LIN {X 0,Y 48.24,Z 388.391,A -85,B 0,C 180,E1 2305.987,E2 2305.987} C_VEL
LIN {X 0,Y 47.995,Z 386.728,A -85,B 0,C 180,E1 2293.212,E2 2293.212} C_VEL
LIN {X 0,Y 47.942,Z 386.734,A -85,B 0,C 180,E1 2285.605,E2 2285.605} C_VEL
LIN {X 0,Y 48.065,Z 388.198,A -85,B 0,C 180,E1 2273.271,E2 2273.271} C_VEL
LIN {X 0,Y 48.162,Z 390.984,A -85,B 0,C 180,E1 2263.191,E2 2263.191} C_VEL
LIN {X 0,Y 48.329,Z 394.762,A -85,B 0,C 180,E1 2253.549,E2 2253.549} C_VEL
LIN {X 0,Y 48.549,Z 397.17,A -85,B 0,C 180,E1 2249.106,E2 2249.106} C_VEL
LIN {X 0,Y 51.151,Z 404.838,A -85,B 0,C 180,E1 2241.844,E2 2241.844} C_VEL
LIN {X 0,Y 54.003,Z 415.083,A -85,B 0,C 180,E1 2234.763,E2 2234.763} C_VEL
LIN {X 0,Y 55.667,Z 422.65,A -85,B 0,C 180,E1 2230.703,E2 2230.703} C_VEL
LIN {X 0,Y 54.802,Z 430.507,A -85,B 0,C 180,E1 2228.864,E2 2228.864} C_VEL
LIN {X 0,Y 53.242,Z 438.053,A -85,B 0,C 180,E1 2227.642,E2 2227.642} C_VEL
LIN {X 0,Y 48.446,Z 450.662,A -85,B 0,C 180,E1 2227.18,E2 2227.18} C_VEL
LIN {X 0,Y 44.463,Z 461.245,A -85,B 0,C 180,E1 2226.637,E2 2226.637} C_VEL
LIN {X 0,Y 43.601,Z 464.496,A -85,B 0,C 180,E1 2226.11,E2 2226.11} C_VEL
LIN {X 0,Y 27.533,Z 552.093,A -85,B 0,C 180,E1 2196.046,E2 2196.046} C_VEL
LIN {X 0,Y 24.945,Z 570.876,A -85,B 0,C 180,E1 2182.47,E2 2182.47} C_VEL
LIN {X 0,Y 23.958,Z 589.422,A -85,B 0,C 180,E1 2162.358,E2 2162.358} C_VEL
LIN {X 0,Y 26.267,Z 606.51,A -85,B 0,C 180,E1 2139.933,E2 2139.933} C_VEL
LIN {X 0,Y 32.018,Z 621.738,A -85,B 0,C 180,E1 2121.318,E2 2121.318} C_VEL
LIN {X 0,Y 40.445,Z 635.298,A -85,B 0,C 180,E1 2107.682,E2 2107.682} C_VEL
LIN {X 0,Y 42.578,Z 638.028,A -85,B 0,C 180,E1 2105.277,E2 2105.277} C_VEL
LIN {X 0,Y 41.554,Z 636.131,A -85,B 0,C 180,E1 2095.677,E2 2095.677} C_VEL
LIN {X 0,Y 35.512,Z 623.919,A -85,B 0,C 180,E1 2080.559,E2 2080.559} C_VEL
LIN {X 0,Y 32.444,Z 609.204,A -85,B 0,C 180,E1 2061.953,E2 2061.953} C_VEL
LIN {X 0,Y 32.629,Z 593.396,A -85,B 0,C 180,E1 2044.611,E2 2044.611} C_VEL
LIN {X 0,Y 34.879,Z 576.253,A -85,B 0,C 180,E1 2030.917,E2 2030.917} C_VEL
LIN {X 0,Y 37.359,Z 559.844,A -85,B 0,C 180,E1 2022.08,E2 2022.08} C_VEL
LIN {X 0,Y 54.584,Z 458.036,A -85,B 0,C 180,E1 1994.856,E2 1994.856} C_VEL
LIN {X 0,Y 57.147,Z 444.741,A -85,B 0,C 180,E1 1992.583,E2 1992.583} C_VEL
LIN {X 0,Y 51.317,Z 423.47,A -85,B 0,C 180,E1 1981.202,E2 1981.202} C_VEL
LIN {X 0,Y 48.036,Z 411.58,A -85,B 0,C 180,E1 1972.542,E2 1972.542} C_VEL
LIN {X 0,Y 45.533,Z 403.648,A -85,B 0,C 180,E1 1964.578,E2 1964.578} C_VEL
LIN {X 0,Y 43.876,Z 399.155,A -85,B 0,C 180,E1 1958.128,E2 1958.128} C_VEL
LIN {X 0,Y 42.596,Z 395.62,A -85,B 0,C 180,E1 1951.259,E2 1951.259} C_VEL
LIN {X 0,Y 42.527,Z 393.676,A -85,B 0,C 180,E1 1942.342,E2 1942.342} C_VEL
LIN {X 0,Y 42.574,Z 392.5,A -85,B 0,C 180,E1 1931.102,E2 1931.102} C_VEL
LIN {X 0,Y 42.405,Z 392.941,A -85,B 0,C 180,E1 1921.952,E2 1921.952} C_VEL
LIN {X 0,Y 42.361,Z 394.215,A -85,B 0,C 180,E1 1913.048,E2 1913.048} C_VEL
LIN {X 0,Y 42.382,Z 396.715,A -85,B 0,C 180,E1 1903.826,E2 1903.826} C_VEL
LIN {X 0,Y 44.543,Z 403.317,A -85,B 0,C 180,E1 1893.368,E2 1893.368} C_VEL
LIN {X 0,Y 46.591,Z 410.788,A -85,B 0,C 180,E1 1885.683,E2 1885.683} C_VEL
LIN {X 0,Y 49.259,Z 423.025,A -85,B 0,C 180,E1 1876.785,E2 1876.785} C_VEL
LIN {X 0,Y 49.308,Z 425.298,A -85,B 0,C 180,E1 1875.841,E2 1875.841} C_VEL
LIN {X 0,Y 45.951,Z 454.046,A -85,B 0,C 180,E1 1868.101,E2 1868.101} C_VEL
LIN {X 0,Y 43.601,Z 464.496,A -85,B 0,C 180,E1 1866.11,E2 1866.11} C_VEL
LIN {X 0,Y 41.115,Z 471.832,A -85,B 0,C 180,E1 1865.327,E2 1865.327} C_VEL
LIN {X 0,Y 31.597,Z 490.821,A -85,B 0,C 180,E1 1865.89,E2 1865.89} C_VEL
LIN {X 0,Y 29.543,Z 497.125,A -85,B 0,C 180,E1 1864.731,E2 1864.731} C_VEL
LIN {X 0,Y 19.494,Z 551.927,A -85,B 0,C 180,E1 1837.008,E2 1837.008} C_VEL
LIN {X 0,Y 17.062,Z 570.883,A -85,B 0,C 180,E1 1816.987,E2 1816.987} C_VEL
LIN {X 0,Y 17.486,Z 589.206,A -85,B 0,C 180,E1 1788.408,E2 1788.408} C_VEL
LIN {X 0,Y 21.991,Z 605.483,A -85,B 0,C 180,E1 1763.722,E2 1763.722} C_VEL
LIN {X 0,Y 29.969,Z 620.693,A -85,B 0,C 180,E1 1746.758,E2 1746.758} C_VEL
LIN {X 0,Y 35.281,Z 628.282,A -85,B 0,C 180,E1 1740.008,E2 1740.008} C_VEL
LIN {X 0,Y 28.789,Z 615.343,A -85,B 0,C 180,E1 1723.361,E2 1723.361} C_VEL
LIN {X 0,Y 25.584,Z 600.444,A -85,B 0,C 180,E1 1702.155,E2 1702.155} C_VEL
LIN {X 0,Y 25.863,Z 584.647,A -85,B 0,C 180,E1 1682.379,E2 1682.379} C_VEL
LIN {X 0,Y 28.227,Z 567.277,A -85,B 0,C 180,E1 1667.031,E2 1667.031} C_VEL
LIN {X 0,Y 30.684,Z 549.124,A -85,B 0,C 180,E1 1656.954,E2 1656.954} C_VEL
LIN {X 0,Y 50.186,Z 446.163,A -85,B 0,C 180,E1 1628.033,E2 1628.033} C_VEL
LIN {X 0,Y 45.374,Z 425.879,A -85,B 0,C 180,E1 1615.199,E2 1615.199} C_VEL
LIN {X 0,Y 42.764,Z 414.063,A -85,B 0,C 180,E1 1604.9,E2 1604.9} C_VEL
LIN {X 0,Y 40.984,Z 406.926,A -85,B 0,C 180,E1 1595.903,E2 1595.903} C_VEL
LIN {X 0,Y 39.565,Z 402.216,A -85,B 0,C 180,E1 1586.248,E2 1586.248} C_VEL
LIN {X 0,Y 38.742,Z 400.308,A -85,B 0,C 180,E1 1577.885,E2 1577.885} C_VEL
LIN {X 0,Y 38.414,Z 399.313,A -85,B 0,C 180,E1 1568.644,E2 1568.644} C_VEL
LIN {X 0,Y 38.75,Z 400.945,A -85,B 0,C 180,E1 1556.417,E2 1556.417} C_VEL
LIN {X 0,Y 39.502,Z 403.672,A -85,B 0,C 180,E1 1548.052,E2 1548.052} C_VEL
LIN {X 0,Y 40.709,Z 409.001,A -85,B 0,C 180,E1 1538.998,E2 1538.998} C_VEL
LIN {X 0,Y 42.073,Z 416.377,A -85,B 0,C 180,E1 1530.739,E2 1530.739} C_VEL
LIN {X 0,Y 43.608,Z 426.272,A -85,B 0,C 180,E1 1522.724,E2 1522.724} C_VEL
LIN {X 0,Y 39.642,Z 454.041,A -85,B 0,C 180,E1 1514.795,E2 1514.795} C_VEL
LIN {X 0,Y 29.543,Z 497.125,A -85,B 0,C 180,E1 1504.731,E2 1504.731} C_VEL
LIN {X 0,Y 27.058,Z 504.449,A -85,B 0,C 180,E1 1503.28,E2 1503.28} C_VEL
LIN {X 0,Y 17.518,Z 523.419,A -85,B 0,C 180,E1 1502.304,E2 1502.304} C_VEL
LIN {X 0,Y 15.546,Z 529.721,A -85,B 0,C 180,E1 1499.393,E2 1499.393} C_VEL
LIN {X 0,Y 10.497,Z 558.063,A -85,B 0,C 180,E1 1469.129,E2 1469.129} C_VEL
LIN {X 0,Y 10.233,Z 577.5,A -85,B 0,C 180,E1 1425.778,E2 1425.778} C_VEL
LIN {X 0,Y 15.654,Z 595.112,A -85,B 0,C 180,E1 1392.657,E2 1392.657} C_VEL
LIN {X 0,Y 24.147,Z 610.841,A -85,B 0,C 180,E1 1377.02,E2 1377.02} C_VEL
LIN {X 0,Y 24.651,Z 611.601,A -85,B 0,C 180,E1 1376.05,E2 1376.05} C_VEL
LIN {X 0,Y 19.626,Z 596.789,A -85,B 0,C 180,E1 1352.942,E2 1352.942} C_VEL
LIN {X 0,Y 18.717,Z 580.526,A -85,B 0,C 180,E1 1326.405,E2 1326.405} C_VEL
LIN {X 0,Y 20.684,Z 563.721,A -85,B 0,C 180,E1 1306.533,E2 1306.533} C_VEL
LIN {X 0,Y 24.177,Z 538.894,A -85,B 0,C 180,E1 1289.754,E2 1289.754} C_VEL
LIN {X 0,Y 43.519,Z 447.587,A -85,B 0,C 180,E1 1262.241,E2 1262.241} C_VEL
LIN {X 0,Y 39.992,Z 428.612,A -85,B 0,C 180,E1 1247.882,E2 1247.882} C_VEL
LIN {X 0,Y 38.408,Z 418.024,A -85,B 0,C 180,E1 1237.038,E2 1237.038} C_VEL
LIN {X 0,Y 37.468,Z 411.862,A -85,B 0,C 180,E1 1227.77,E2 1227.77} C_VEL
LIN {X 0,Y 36.977,Z 408.929,A -85,B 0,C 180,E1 1220.677,E2 1220.677} C_VEL
LIN {X 0,Y 36.567,Z 407.094,A -85,B 0,C 180,E1 1209.511,E2 1209.511} C_VEL
LIN {X 0,Y 36.611,Z 408.513,A -85,B 0,C 180,E1 1199.13,E2 1199.13} C_VEL
LIN {X 0,Y 36.866,Z 410.647,A -85,B 0,C 180,E1 1192.82,E2 1192.82} C_VEL
LIN {X 0,Y 37.285,Z 414.995,A -85,B 0,C 180,E1 1185.206,E2 1185.206} C_VEL
LIN {X 0,Y 37.971,Z 422.73,A -85,B 0,C 180,E1 1176.129,E2 1176.129} C_VEL
LIN {X 0,Y 38.339,Z 428.6,A -85,B 0,C 180,E1 1171.033,E2 1171.033} C_VEL
LIN {X 0,Y 33.997,Z 453.882,A -85,B 0,C 180,E1 1163.709,E2 1163.709} C_VEL
LIN {X 0,Y 15.546,Z 529.721,A -85,B 0,C 180,E1 1139.393,E2 1139.393} C_VEL
LIN {X 0,Y 13.154,Z 537.031,A -85,B 0,C 180,E1 1135.253,E2 1135.253} C_VEL
LIN {X 0,Y 3.16,Z 556.731,A -85,B 0,C 180,E1 1100.557,E2 1100.557} C_VEL
LIN {X 0,Y 2.925,Z 561.897,A -85,B 0,C 180,E1 1059.568,E2 1059.568} C_VEL
LIN {X 0,Y 9.168,Z 579.993,A -85,B 0,C 180,E1 1011.793,E2 1011.793} C_VEL
LIN {X 0,Y 13.89,Z 589.571,A -85,B 0,C 180,E1 1005.16,E2 1005.16} C_VEL
LIN {X 0,Y 11.881,Z 572.674,A -85,B 0,C 180,E1 967.955,E2 967.955} C_VEL
LIN {X 0,Y 13.528,Z 556.998,A -85,B 0,C 180,E1 941.938,E2 941.938} C_VEL
LIN {X 0,Y 37.368,Z 449.245,A -85,B 0,C 180,E1 894.831,E2 894.831} C_VEL
LIN {X 0,Y 35.318,Z 431.366,A -85,B 0,C 180,E1 878.711,E2 878.711} C_VEL
LIN {X 0,Y 34.83,Z 421.783,A -85,B 0,C 180,E1 867.22,E2 867.22} C_VEL
LIN {X 0,Y 34.755,Z 417.397,A -85,B 0,C 180,E1 859.423,E2 859.423} C_VEL
LIN {X 0,Y 34.722,Z 415.741,A -85,B 0,C 180,E1 854.851,E2 854.851} C_VEL
LIN {X 0,Y 34.669,Z 414.985,A -85,B 0,C 180,E1 848.899,E2 848.899} C_VEL
LIN {X 0,Y 34.553,Z 416.368,A -85,B 0,C 180,E1 841.108,E2 841.108} C_VEL
LIN {X 0,Y 34.334,Z 420.433,A -85,B 0,C 180,E1 833.363,E2 833.363} C_VEL
LIN {X 0,Y 34.168,Z 427.831,A -85,B 0,C 180,E1 824.174,E2 824.174} C_VEL
LIN {X 0,Y 34.025,Z 430.755,A -85,B 0,C 180,E1 821.623,E2 821.623} C_VEL
LIN {X 0,Y 29.34,Z 453.762,A -85,B 0,C 180,E1 815.604,E2 815.604} C_VEL
LIN {X 0,Y 3.767,Z 549.95,A -85,B 0,C 180,E1 771.651,E2 771.651} C_VEL
LIN {X 0,Y 2.925,Z 561.897,A -85,B 0,C 180,E1 699.568,E2 699.568} C_VEL
LIN {X 0,Y 2.549,Z 561.961,A -85,B 0,C 180,E1 680.822,E2 680.822} C_VEL
LIN {X 0,Y 2.311,Z 560.057,A -85,B 0,C 180,E1 631.507,E2 631.507} C_VEL
LIN {X 0,Y 3.836,Z 554.913,A -85,B 0,C 180,E1 583.045,E2 583.045} C_VEL
LIN {X 0,Y 7.562,Z 543.659,A -85,B 0,C 180,E1 557.848,E2 557.848} C_VEL
LIN {X 0,Y 8.341,Z 540.505,A -85,B 0,C 180,E1 553.983,E2 553.983} C_VEL
LIN {X 0,Y 31.914,Z 450.165,A -85,B 0,C 180,E1 524.234,E2 524.234} C_VEL
LIN {X 0,Y 31.686,Z 433.671,A -85,B 0,C 180,E1 506.649,E2 506.649} C_VEL
LIN {X 0,Y 32.357,Z 425.561,A -85,B 0,C 180,E1 495.535,E2 495.535} C_VEL
LIN {X 0,Y 32.727,Z 423.005,A -85,B 0,C 180,E1 489.892,E2 489.892} C_VEL
LIN {X 0,Y 32.636,Z 423.325,A -85,B 0,C 180,E1 487.453,E2 487.453} C_VEL
LIN {X 0,Y 31.789,Z 427.902,A -85,B 0,C 180,E1 479.938,E2 479.938} C_VEL
LIN {X 0,Y 31.082,Z 432.7,A -85,B 0,C 180,E1 474.662,E2 474.662} C_VEL
LIN {X 0,Y 26.246,Z 453.556,A -85,B 0,C 180,E1 470.94,E2 470.94} C_VEL
LIN {X 0,Y 4.449,Z 548.941,A -85,B 0,C 180,E1 561.616,E2 561.616} C_VEL
LIN {X 0,Y 5.592,Z 556.043,A -85,B 0,C 180,E1 584.45,E2 584.45} C_VEL
LIN {X 0,Y 8.341,Z 540.505,A -85,B 0,C 180,E1 553.983,E2 553.983} C_VEL
LIN {X 0,Y 11.641,Z 541.048,A -85,B 0,C 180,E1 541.61,E2 541.61} C_VEL
LIN {X 0,Y 11.641,Z 565.756,A -85,B 0,C 180,E1 541.61,E2 541.61} C_VEL
LIN {X 0,Y 15.989,Z 565.756,A -85,B 0,C 180,E1 507.842,E2 507.842} C_VEL
LIN {X 0,Y 15.989,Z 535.345,A -85,B 0,C 180,E1 507.842,E2 507.842} C_VEL
LIN {X 0,Y 15.989,Z 494.766,A -85,B 0,C 180,E1 507.842,E2 507.842} C_VEL
LIN {X 0,Y 16.063,Z 494.223,A -85,B 0,C 180,E1 507.877,E2 507.877} C_VEL
LIN {X 0,Y 27.773,Z 451.482,A -85,B 0,C 180,E1 510.546,E2 510.546} C_VEL
LIN {X 0,Y 29.538,Z 436.414,A -85,B 0,C 180,E1 492.812,E2 492.812} C_VEL
LIN {X 0,Y 29.966,Z 434.28,A -85,B 0,C 180,E1 489.649,E2 489.649} C_VEL
LIN {X 0,Y 25.291,Z 453.25,A -85,B 0,C 180,E1 488.718,E2 488.718} C_VEL
LIN {X 0,Y 16.063,Z 494.223,A -85,B 0,C 180,E1 507.877,E2 507.877} C_VEL
LIN {X 0,Y 16.086,Z 495.48,A -85,B 0,C 180,E1 509.459,E2 509.459} C_VEL
LIN {X 0,Y 16.086,Z 779,A -85,B 0,C 180,E1 509.459,E2 509.459} C_VEL
LIN {X 0,Y 16.086,Z 779,A -85,B 0,C 180,E1 509.459,E2 509.459}

QRS_NEXT_CUT()

QRS_NEXT()
QRS_HOME()

END
